//Note: the execution time is monitored by a base Fb timer. Therefore a timeout may occur. This behavior is configurable.
END_METHOD

METHOD PRIVATE FINAL M_FinishCommand
VAR 
	strLogMsg : STRING;	
END_VAR
IF localCmd.Control = cAbort AND bAbortionAllowed THEN		//Command was aborted by host
	localRes.Status := cFinAbrtd;

ELSIF localRes.Error = GVL.ERR_NO_ERROR THEN					//executed without error
	localRes.Status := cFinOk;
	
	//Log data
		M_Log(	LogLevel 	:= eLogLevel.TRACE, 
				strMethod 	:= 'M_FinishCommand',
				strLogMsg 	:= '|ADS - command finished successfully by SPS');	
ELSE
	localRes.Status := cFinErr;								//executed with error
	//Log data
		strLogMsg := CONCAT('|ADS - command finished faulty by SPS with ErrorId: ', WORD_TO_STRING(localRes.Error));
	
		M_Log(	LogLevel 	:= eLogLevel.TRACE, 
				strMethod 	:= 'M_FinishCommand',
				strLogMsg 	:= strLogMsg);				
END_IF

bCmdEnabledByIntern := TRUE;
eState := eCmdProcessing._RECEIVING;
END_METHOD

METHOD PROTECTED FINAL M_Log
VAR_INPUT
	strMethod 	: STRING(40);
	strLogMsg 	: STRING;
	LogLevel 	: eLogLevel;
END_VAR
VAR
	strCaller : STRING := 'FB_wCMD_Handler_Base.';
END_VAR
IF NOT GVL_AdsInterface.bLoggingOnOff_IncomingAds THEN 
	RETURN;
END_IF

strCaller := CONCAT(strInstanceName, '.');
strCaller := CONCAT(strCaller, strMethod);

//If Logging.prg is not available in project or to deactivate logging completely, just comment the following line out!
	Logging.Debug(strCaller, strLogMsg);
END_METHOD

METHOD PRIVATE FINAL M_ReceiveCommand
IF localCmd.Control = cRcv THEN
		
	//Delete result structure variable
		MEMSET(destaddr := ADR(localRes), fillbyte:=0, n:= SIZEOF(localRes));
		localres.ErrorComp 	:= wCompId;
		localres.Error 		:= GVL.ERR_NO_ERROR;
	
	//Set result struct to state RECEIVED even if there could be errors
		localRes.Status := cRcvd;
	
	//Check if command is currently blocked
	IF bCmdEnabledByExtern AND bCmdEnabledByIntern THEN
		bCmdEnabledByIntern := FALSE;
		
	ELSIF NOT bCmdEnabledByIntern THEN		
		localRes.Error := GVL_AdsInterface_ERROR_IDS.ERR_ITF_COMMAND_CAN_NOT_BE_ENABLED_THUS_INTERNALLY_DISABLED + GVL_AdsInterface.wErrorIdOffset_IncomingAds;
		
	ELSIF NOT bCmdEnabledByExtern THEN
		localRes.Error := GVL_AdsInterface_ERROR_IDS.ERR_ITF_COMMAND_CAN_NOT_BE_ENABLED_THUS_EXTERNALLY_DISABLED + GVL_AdsInterface.wErrorIdOffset_IncomingAds;
		
	ELSE
		localRes.Error := GVL_AdsInterface_ERROR_IDS.ERR_ITF_INCOMING_COMMAND_IS_BLOCKED + GVL_AdsInterface.wErrorIdOffset_IncomingAds;
		
	END_IF
	
	//Check incomming command parameter for correctness
		IF localCmd.Version 	<> wVersion 			THEN localRes.Error := GVL_AdsInterface_ERROR_IDS.ERR_ITF_INCOMING_COMMAND_HAS_WRONG_VERSION + GVL_AdsInterface.wErrorIdOffset_IncomingAds; 			END_IF;
		IF iParTyp 	<> PAR_TYPE_REGARDLESS THEN 
			IF localCmd.ParaCount 	<> iParCount 	THEN localRes.Error := GVL_AdsInterface_ERROR_IDS.ERR_ITF_INCOMING_COMMAND_HAS_WRONG_PARAMETER_COUNT + GVL_AdsInterface.wErrorIdOffset_IncomingAds; 	END_IF;
			IF localCmd.ParaTyp	 	<> iParTyp 		THEN localRes.Error := GVL_AdsInterface_ERROR_IDS.ERR_ITF_INCOMING_COMMAND_HAS_WRONG_PARAMETER_TYP + GVL_AdsInterface.wErrorIdOffset_IncomingAds; 	END_IF;				
		END_IF
END_IF
END_METHOD

PROPERTY PUBLIC final P_EnabledInternally : bool
GET
P_EnabledInternally := bCmdEnabledByIntern;
END_GET
END_PROPERTY

END_FUNCTION_BLOCK

// AdsInterface/FB_SendAdsDocCmd_Base
//Author: 				Walther Ronny
//Version:				1.0
//Last change:			14.04.16
//See Release notes at the bottom
//{attribute 'hide_all_locals'}
{attribute 'reflection'}
FUNCTION_BLOCK PUBLIC FB_SendAdsDocCmd_Base				//Base Fb for handling of ADS communication of type TwRes and TwCmd
VAR_OUTPUT
	bDone,
	bError : BOOL;
	ErrorMsg : sErrorMsg;
    {attribute 'instance-path'}
    {attribute 'no_init'}
    sPath  : STRING;
END_VAR 
VAR_INPUT		
	Instanz: BYTE; 										//Instanz counter 
	pCmd : POINTER TO TxCmdRes;							//Pointer to incomming command structure from host
	pRes : POINTER TO TxCmdRes;							//Pointer to outgoing result structure from SPS
END_VAR
VAR
	wCompId : WORD;		//Component ID
//Command configuration which has to be set by instantiated Fb - 	MUST !
	wVersion : 				WORD := 0;	//Expected version of incomming command
	iParTyp1: 				BYTE := 0;	//Expected parameter type of incomming command, PAR_TYPE_REGARDLESS will switch test off
	iParCount1 : 			BYTE := 0;	//Expected parameter count of incomming command
	iParTyp2 : 				BYTE := 0;	//Expected parameter type of incomming command, PAR_TYPE_REGARDLESS will switch test off
	iParCount2 : 			BYTE := 0;	//Expected parameter count of incomming command
	
//Command configuration which can be set by instantiated Fb - 	OPTIONALLY !
	tExecutionTimeout : 	TIME := ADS_EXECUTION_TIMEOUT; 	//Timeout while Execution running. T#0s equals off
	
	bStartSendingData : BOOL := FALSE;	//flag to indicate that data can be sent				

//This variable can be used to hold the state of the derived M_ExecuteCommand() 
	iHelpState : UINT := 0;	//optional help variable to create a statemachine inside derive M_ExecuteCommand()
	
//Local Command and result structure objects - Will be read and written by base Fb and derived "M_ExecuteCommand()" method
	localRes: TdocRes;
	localCmd: TdocCmd;	
	
//Internal variables of base Fb - DO NOT CHANGE!	
	bCmdEnabledByExtern,								//Command is enabled/disabled  externally (by MainFSM)
	bCmdEnabledByIntern : 	BOOL:= TRUE;				//Command is enabled/disabled  internally during execution
		
	eState: eSendCmdProcessing := eSendCmdProcessing._IDLE;	//Current internal state of the base Fb		
	TimerExecutionTimeout : ton;						// Timer for Execution timeout
END_VAR
VAR CONSTANT
	//Command parameter types
	PAR_TYPE_REGARDLESS :		BYTE := 0;			//if this type is set, the parameter type will be not checked
	PAR_TYPE_ANSICHAR : 		BYTE := 16#41;
	PAR_TYPE_SHORTINT : 		BYTE := 16#53;
	PAR_TYPE_WIDECHAR : 		BYTE := 16#43;
	PAR_TYPE_SMALLINT : 		BYTE := 16#4D;
	PAR_TYPE_LONGINT : 			BYTE := 16#49;
	PAR_TYPE_LONGWORD : 		BYTE := 16#4C;
	PAR_TYPE_WORD : 			BYTE := 16#57;		//Standard parameter type
	PAR_TYPE_BIT : 				BYTE := 16#58;
	
	ADS_EXECUTION_TIMEOUT :		TIME := T#10S;		//Timeout while derived Execution method is executed. T#0S equals OFF

		// command
	cAbort:						WORD := 0;			// command abort				
	cRcv:						WORD := 1;			// command receive				
	cExec:						WORD := 2;			// command start				
	// result
	cIdle: 						WORD := 0;      	// not  defined					
	cRcvd:						WORD := 1;      	// command received 			
	cActive:					WORD := 2;			// command active started 		
	cFinOk:						WORD := 4;			// command finished ok			
	cFinAbrtd:					WORD := 5;			// command aborted				
	cFinErr:					WORD := 6;			// command finished error		
END_VAR

(*
Release notes:
1.0 	Walther Ronny, 14.04.16
		- Initial version
*)

ErrorMsg.sFunctionName := 'FB_SendAdsDocCmd_Base';

	wCompId := GVL_AdsInterface.wCompId_OutgoingAds;
	
//Create local copy of actual result struct
	localRes := pRes^.docRes;

CASE eState OF
	
	eSendCmdProcessing._IDLE :
	
			//reset flags
				bError 	:= FALSE;
				bDone	:= FALSE;
				
			//reset timeout timer
				TimerExecutionTimeout.IN := FALSE;
				
			//Check for start sending flag	
				IF bStartSendingData THEN
					bStartSendingData := FALSE;
					
					//disable cmd
						bCmdEnabledByIntern := FALSE;
						
					//Set receive parameter
						localCmd.Control := cRcv;
						
					//Set local data to outgoing command struct					
						pCmd^.docCmd := localCmd;
					
					eState := eSendCmdProcessing._SENDING;
					Logging.Trace('FB_SendAdsDocCmd_Base','State change: IDLE - SENDING');
				END_IF
				
	eSendCmdProcessing._SENDING :
	
			IF localRes.Status = cRcvd THEN
				
				//Start command
					pCmd^.docCmd.Control := cExec;
					
				eState := eSendCmdProcessing._STARTING;
				Logging.Trace('FB_SendAdsDocCmd_Base','State change: SENDING - STARTING');
			END_IF
			
	eSendCmdProcessing._STARTING :
					
			//start timeout timer
				TimerExecutionTimeout(IN := TRUE, PT := tExecutionTimeout);
				
			//Wait for result state	to change
				IF localRes.Status <> cRcvd THEN				
					eState := eSendCmdProcessing._EXECUTING;
					Logging.Trace('FB_SendAdsDocCmd_Base','State change: STARTING - EXECUTING');
				END_IF
			
	eSendCmdProcessing._EXECUTING :
	
			IF localRes.Status = cFinOk THEN
				eState := eSendCmdProcessing._DONE;
				Logging.Trace('FB_SendAdsDocCmd_Base','State change: EXECUTING - DONE (cFinOK)');
			ELSIF localRes.Status = cFinAbrtd THEN
				bError 				:= TRUE;
				ErrorMsg.wComponent := wCompId;
				ErrorMsg.wErrorNo 	:= GVL_AdsInterface_ERROR_IDS.ERR_ITF_COMMAND_WAS_ABORTED_BY_HOST_DURING_EXECUTION + GVL_AdsInterface.wErrorIdOffset_OutgoingAds;
				
				eState := eSendCmdProcessing._DONE;
				Logging.Trace('FB_SendAdsDocCmd_Base','State change: EXECUTING - DONE (cFinAbrtd)');
			ELSIF localRes.Status = cFinErr THEN
				bError 				:= TRUE;
				ErrorMsg.wComponent := wCompId;
				ErrorMsg.wErrorNo 	:= localRes.Error + GVL_AdsInterface.wErrorIdOffset_OutgoingAds;
				
				eState := eSendCmdProcessing._DONE;
				Logging.Trace('FB_SendAdsDocCmd_Base','State change: EXECUTING - DONE (cFinErr)');
			ELSIF TimerExecutionTimeout.Q AND tExecutionTimeout <> T#0S THEN
				bError 				:= TRUE;
				ErrorMsg.wComponent := wCompId;
				ErrorMsg.wErrorNo 	:= GVL_AdsInterface_ERROR_IDS.ERR_ITF_COMMAND_EXECUTION_TIMEOUT + GVL_AdsInterface.wErrorIdOffset_OutgoingAds;
					
				eState := eSendCmdProcessing._DONE; 
				Logging.Trace('FB_SendAdsDocCmd_Base','State change: EXECUTING - DONE (timeout)');		
			END_IF
			
	eSendCmdProcessing._DONE : 
	
			//reset timeout timer
				TimerExecutionTimeout.IN := FALSE;
				
			bCmdEnabledByIntern := TRUE;
			
			bDone:= TRUE;
			
			//Check for start sending flag	
				IF bStartSendingData THEN
					eState := eSendCmdProcessing._IDLE;
					
				END_IF

END_CASE

TimerExecutionTimeout();

METHOD PUBLIC M_EnableCmd
VAR_INPUT
	bEnable : BOOL := FALSE; //TRUE = Command is enabled, FALSE = Command i disabled
END_VAR
bCmdEnabledByExtern := bEnable;
END_METHOD

METHOD PUBLIC M_SendCmd				//Sending an ADS command
VAR_INPUT
	docCmdData 		: TdocCmd; 		//command structure to be sent
END_VAR
VAR_OUTPUT
	bMethodError 	: BOOL;			//indicates an error
	MethodErrorMsg 	: sErrorMsg;	//describes an error
END_VAR
//Check command state
	IF eState = eSendCmdProcessing._IDLE OR eState = eSendCmdProcessing._DONE THEN
	
	//Reset fb output state
		bDone := FALSE;
		bError := FALSE;
		ErrorMsg.wComponent := wCompId;
		ErrorMsg.wErrorNo 	:= GVL.ERR_NO_ERROR;
		
		M_SetLocalData(pDocCmd := ADR(docCmdData), bError => bMethodError, ErrorMsg => MethodErrorMsg);
		
		IF NOT bMethodError THEN
			//start sending data
				bStartSendingData := TRUE;
				
		END_IF
		
	ELSE //e.g. still activ...
		bMethodError := TRUE;
		MethodErrorMsg.wComponent := wCompId;
		MethodErrorMsg.wErrorNo	:= GVL_AdsInterface_ERROR_IDS.ERR_ITF_WRONG_FB_STATE_TO_SEND_COMMAND + GVL_AdsInterface.wErrorIdOffset_OutgoingAds;
		
	END_IF
END_METHOD

METHOD PRIVATE M_SetLocalData
VAR_INPUT
	pDocCmd : pointer to TdocCmd;
END_VAR
VAR_OUTPUT
	bError : 	BOOL;
	ErrorMsg : 	sErrorMsg;
END_VAR
	//Delete result structure variable
		MEMSET(destaddr := ADR(localRes), fillbyte:=0, n:= SIZEOF(localRes));
	
	//Check if command is currently blocked
	IF bCmdEnabledByExtern AND bCmdEnabledByIntern THEN
		ErrorMsg.wErrorNo := GVL.ERR_NO_ERROR;
		bCmdEnabledByIntern := FALSE;
		
	ELSIF NOT bCmdEnabledByIntern THEN		
		ErrorMsg.wErrorNo := GVL_AdsInterface_ERROR_IDS.ERR_ITF_COMMAND_CAN_NOT_BE_ENABLED_THUS_INTERNALLY_DISABLED + GVL_AdsInterface.wErrorIdOffset_OutgoingAds;
		
	ELSIF NOT bCmdEnabledByExtern THEN
		ErrorMsg.wErrorNo := GVL_AdsInterface_ERROR_IDS.ERR_ITF_COMMAND_CAN_NOT_BE_ENABLED_THUS_EXTERNALLY_DISABLED + GVL_AdsInterface.wErrorIdOffset_OutgoingAds;
		
	ELSE
		ErrorMsg.wErrorNo := GVL_AdsInterface_ERROR_IDS.ERR_ITF_INCOMING_COMMAND_IS_BLOCKED + GVL_AdsInterface.wErrorIdOffset_OutgoingAds;
		
	END_IF
	
	//Check incomming command parameter for correctness
		IF pDocCmd^.Version 	<> wVersion 			THEN ErrorMsg.wErrorNo := GVL_AdsInterface_ERROR_IDS.ERR_ITF_INCOMING_COMMAND_HAS_WRONG_VERSION + GVL_AdsInterface.wErrorIdOffset_OutgoingAds; 		END_IF;
			
		IF iParTyp1 	<> PAR_TYPE_REGARDLESS 	THEN 
			IF pDocCmd^.ParaCount1 	<> iParCount1 	THEN ErrorMsg.wErrorNo := GVL_AdsInterface_ERROR_IDS.ERR_ITF_INCOMING_COMMAND_HAS_WRONG_PARAMETER_COUNT + GVL_AdsInterface.wErrorIdOffset_OutgoingAds; 	END_IF;
			IF pDocCmd^.ParaTyp1	<> iParTyp1		THEN ErrorMsg.wErrorNo := GVL_AdsInterface_ERROR_IDS.ERR_ITF_INCOMING_COMMAND_HAS_WRONG_PARAMETER_TYP + GVL_AdsInterface.wErrorIdOffset_OutgoingAds; 	END_IF;	
		END_IF;	
		
		IF iParTyp2 	<> PAR_TYPE_REGARDLESS THEN
			IF pDocCmd^.ParaCount2 	<> iParCount2 	THEN ErrorMsg.wErrorNo := GVL_AdsInterface_ERROR_IDS.ERR_ITF_INCOMING_COMMAND_HAS_WRONG_PARAMETER_COUNT + GVL_AdsInterface.wErrorIdOffset_OutgoingAds; 	END_IF;			
			IF pDocCmd^.ParaTyp2	<> iParTyp2		THEN ErrorMsg.wErrorNo := GVL_AdsInterface_ERROR_IDS.ERR_ITF_INCOMING_COMMAND_HAS_WRONG_PARAMETER_TYP + GVL_AdsInterface.wErrorIdOffset_OutgoingAds; 	END_IF;	
		END_IF
	ErrorMsg.wComponent := wCompId;
	
	IF ErrorMsg.wErrorNo <> GVL.ERR_NO_ERROR THEN
		bError:= TRUE;
	ELSE
		localCmd := pDocCmd^;	

	END_IF
END_METHOD

PROPERTY PUBLIC P_CommandState : eSendCmdProcessing
GET
P_CommandState := eState;
END_GET
END_PROPERTY

PROPERTY PUBLIC P_EnabledInternally : bool
GET
P_EnabledInternally := bCmdEnabledByIntern;
END_GET
END_PROPERTY

END_FUNCTION_BLOCK

// AdsInterface/FB_wCMD_docCMD_Handler_Base2
//Author: 				Walther Ronny
//Version:				1.6
//Last change:			16.10.2018
//See Release notes at the bottom
//{attribute 'hide_all_locals'}
{attribute 'reflection'}
FUNCTION_BLOCK PUBLIC FB_wCMD_docCMD_Handler_Base2				//Base Fb for handling of ADS communication of type TwRes and TwCmd
VAR_OUTPUT
    {attribute 'instance-path'}
    {attribute 'no_init'}
    sPath  		: STRING; 	//Instance path
	pLogCmdRes 	: POINTER TO ARRAY [0.. LOG_CMDRES_MAX] OF TxCmdRes2Double := ADR(arrLogCmdRes);
	pLogCmdResIndex: POINTER TO UINT := ADR(nLogIndexCmdRes);
END_VAR 
VAR_INPUT		
	Instanz: BYTE; 										//Instanz counter 
	pCmd : POINTER TO TxCmdRes2;						//Pointer to incomming command structure from host
	pRes : POINTER TO TxCmdRes2;						//Pointer to outgoing result structure from SPS
END_VAR
VAR		
	wCompId : WORD;		//Component ID
//Command configuration which has to be set by instantiated Fb - 	MUST !
	wVersion : 				WORD := 0;	//Expected version of incomming command
	iParTyp1 : 				BYTE := 0;	//Expected parameter type of incomming command, PAR_TYPE_REGARDLESS will switch test off
	iParCount1 : 			BYTE := 0;	//Expected parameter count of incomming command
	iParTyp2 : 				BYTE := 0;	//Expected parameter type of incomming command, PAR_TYPE_REGARDLESS will switch test off
	iParCount2 : 			BYTE := 0;	//Expected parameter count of incomming command
		
//Command configuration which can be set by instantiated Fb - 	OPTIONALLY !
	bAbortionAllowed : 		BOOL 		:= TRUE;					//if yes, abortion from host is allowed all the time
	tExecutionTimeout : 	TIME 		:= ADS_EXECUTION_TIMEOUT; 	//Timeout while Execution running. T#0s equals off
	strInstanceName :		STRING(40);								//Name of instance of that base class (used only for logging purposes)
//Flag to indicate that the derived method "M_ExecuteCommand()" finished	
	bExecutionDone : BOOL := FALSE;	//flag to indicate that derived Execution is done				

//This variable can be used to hold the state of the derived M_ExecuteCommand() 
	iHelpState : UINT := 0;	//optional help variable to create a statemachine inside derive M_ExecuteCommand()
	
//Local Command and result structure objects - Will be read and written by base Fb and derived "M_ExecuteCommand()" method
	localRes: TxCmdRes2;//TwRes2;
	localCmd: TxCmdRes2;//TwCmd2;	
	
//Internal variables of base Fb - DO NOT CHANGE!	
	bCmdEnabledByExtern,								//Command is enabled/disabled  externally (by MainFSM)
	bCmdEnabledByIntern : 	BOOL:= TRUE;				//Command is enabled/disabled  internally during execution
		
	eState: eCmdProcessing := eCmdProcessing._RECEIVING;	//Current internal state of the base Fb		
	TimerExecutionTimeout : ton;							// Timer for Execution timeout
	
// log ads communication for debugging	
	nCmpResult, nCmpCommand: DINT;
	nLogIndexCmdRes: UINT;
	arrLogCmdRes: ARRAY [0.. LOG_CMDRES_MAX] OF TxCmdRes2Double;
	
	
END_VAR
VAR CONSTANT
	LOG_CMDRES_MAX:				UINT := 10;
	DATA_LENGT_IN_8byte:		UINT := 7;	

	//Command parameter types
	PAR_TYPE_REGARDLESS :		BYTE := 0;		//if this type is set, the parameter type will be not checked
	PAR_TYPE_ANSICHAR : 		BYTE := 16#41; //8bit
	PAR_TYPE_BYTE : 			BYTE := 16#42; //8bit
	PAR_TYPE_WIDECHAR : 		BYTE := 16#43; //16bit
	PAR_TYPE_FLOAT : 			BYTE := 16#44; //64bit	
	PAR_TYPE_SHORTINT : 		BYTE := 16#53; //8bit	
	PAR_TYPE_SMALLINT : 		BYTE := 16#4D; //16bit
	PAR_TYPE_LONGINT : 			BYTE := 16#49; //32bit
	PAR_TYPE_LONGWORD : 		BYTE := 16#4C; //32bit
	PAR_TYPE_WORD : 			BYTE := 16#57; //16bit
	PAR_TYPE_BIT : 				BYTE := 16#58;
	
	ADS_EXECUTION_TIMEOUT :		TIME := T#30S;		//Timeout while derived Execution method is executed. T#0S equals OFF

		// command
	cAbort:						WORD := 0;			// command abort				
	cRcv:						WORD := 1;			// command receive				
	cExec:						WORD := 2;			// command start				
	// result
	cIdle: 						WORD := 0;      	// not  defined					
	cRcvd:						WORD := 1;      	// command received 			
	cActive:					WORD := 2;			// command active started 		
	cFinOk:						WORD := 4;			// command finished ok			
	cFinAbrtd:					WORD := 5;			// command aborted				
	cFinErr:					WORD := 6;			// command finished error		
END_VAR

(*
Release notes:
1.0 First release. Tested on Holo machine in Munich. 25.01.16
1.1 Aborting modified and tested. Constants included in FB. 26.01.16
1.2 Bug M_ReceiveCommand PARTYP_REGARDLESS fixed
1.3 Walther Ronny, 25.05.16
	- Variable strInstanceName added
	- Method M_Log() added
	- Logging added
1.4 Werner Richter, 19.09.2018
	- FB_wCMD_Handler_Base modifyed to FB_wCMD_Handler_Base2 because communication to host has modified to check data length before sending,
	  use modified data structure TxCmdRes2, check header in state _RECEIVING, modify M_ReceiveCommand, 
      check type in _WAITING_FOR_START, set received flag only if no error
1.5 Werner Richter, 21.09.2018
	- combined FB_wCMD_Handler_Base2 + FB_docCMD_Handler_Base, bAbortionAllowed := TRUE
1.6 Werner Richter, 16.10.2018
	- log ads communication for debugging
*)

//Create local copy of received command struct
	localCmd:=pCmd^;//.wCmd; 

CASE eState OF
	
	eCmdProcessing._RECEIVING: 	//Receiving command
	
				//Check id, thus it might have been changed
					wCompId := GVL_AdsInterface.wCompId_IncomingAds;
				
				IF M_ReceiveCommand() THEN
								
					//Log data
					M_Log(	LogLevel 	:= eLogLevel.TRACE, 
							strMethod 	:= 'FB_wCMD_Handler_Base',
							strLogMsg 	:= '|ADS - command received from host');	
								
					IF localres.wRes.Error = GVL.ERR_NO_ERROR THEN	// check wrong header
								
						localRes.wRes.Status := cRcvd;
						eState := eCmdProcessing._WAITING_FOR_START;					
					ELSE
						
						localRes.wRes.Status := cFinErr;
						
						pCmd^.wCmd.Control := cAbort;			// needed if error in receiving state occured to reset command handshaking
	
						//Log data					
						M_Log(	LogLevel 	:= eLogLevel.TRACE, 
								strMethod 	:= 'M_FinishCommand',
								strLogMsg 	:= CONCAT('|ADS - command finished faulty by SPS with ErrorId: ', WORD_TO_STRING(localRes.wRes.Error)));				
										
						bCmdEnabledByIntern := TRUE;
						eState := eCmdProcessing._RECEIVING;
						
						//reset timer
						TimerExecutionTimeout.IN := FALSE;						
						
					END_IF
					
				END_IF
								
							
				
	eCmdProcessing._WAITING_FOR_START:	//Waiting for Start from Host
					
				IF localCmd.wCmd.Control = cExec THEN //check if the command was started by the host
					//Log data
						M_Log(	LogLevel 	:= eLogLevel.TRACE, 
								strMethod 	:= 'FB_wCMD_Handler_Base',
								strLogMsg 	:= '|ADS - command started by host');	
						
								
					IF localRes.wRes.Error <> GVL.ERR_NO_ERROR THEN //Check if an error during receiving ocurred		
	
						eState := eCmdProcessing._FINISHING;

					ELSIF 	((iParTyp1 <> PAR_TYPE_REGARDLESS) AND ((localCmd.wCmd.ParaCount1 <> iParCount1) OR (localCmd.wCmd.ParaTyp1 <> iParTyp1))) OR
							((iParTyp2 <> PAR_TYPE_REGARDLESS) AND ((localCmd.docCmd.ParaCount2 <> iParCount2) OR (localCmd.docCmd.ParaTyp2 <> iParTyp2))) THEN
					
						// wCmd	+ docCmd	
						IF (iParTyp1 <> PAR_TYPE_REGARDLESS) AND ((localCmd.wCmd.ParaCount1 <> iParCount1) OR (localCmd.wCmd.ParaTyp1 <> iParTyp1)) THEN										
							IF localCmd.wCmd.ParaCount1 <> iParCount1 THEN localRes.wRes.Error := GVL_AdsInterface_ERROR_IDS.ERR_ITF_INCOMING_COMMAND_HAS_WRONG_PARAMETER_COUNT + GVL_AdsInterface.wErrorIdOffset_IncomingAds; 	END_IF;
							IF localCmd.wCmd.ParaTyp1   <> iParTyp1   THEN localRes.wRes.Error := GVL_AdsInterface_ERROR_IDS.ERR_ITF_INCOMING_COMMAND_HAS_WRONG_PARAMETER_TYP + GVL_AdsInterface.wErrorIdOffset_IncomingAds; 	END_IF;										
						END_IF
						
						//docCmd
						IF (iParTyp2 <> PAR_TYPE_REGARDLESS) AND ((localCmd.docCmd.ParaCount2 <> iParCount2) OR (localCmd.docCmd.ParaTyp2 <> iParTyp2)) THEN							
							IF localCmd.docCmd.ParaCount2 <> iParCount2 THEN localRes.wRes.Error := GVL_AdsInterface_ERROR_IDS.ERR_ITF_INCOMING_COMMAND_HAS_WRONG_PARAMETER_COUNT + GVL_AdsInterface.wErrorIdOffset_IncomingAds; 	END_IF;
							IF localCmd.docCmd.ParaTyp2	  <> iParTyp2   THEN localRes.wRes.Error := GVL_AdsInterface_ERROR_IDS.ERR_ITF_INCOMING_COMMAND_HAS_WRONG_PARAMETER_TYP + GVL_AdsInterface.wErrorIdOffset_IncomingAds; 	END_IF;										
						END_IF
						
						eState := eCmdProcessing._FINISHING;

					ELSE
																									
						//Reset variables for derived "M_ExecuteCommand()" method	
							bExecutionDone := FALSE;
							iHelpState := 0;	
						
						localRes.wRes.Status := cActive;					
						eState := eCmdProcessing._EXECUTING;
						
						//start timeout timer
							TimerExecutionTimeout(IN := TRUE, PT := tExecutionTimeout);
					END_IF					
								
					
				END_IF
					
					
	eCmdProcessing._EXECUTING:	//Executing command
			
				IF bExecutionDone THEN //flag will be set by derived method if execution done									
					eState := eCmdProcessing._FINISHING; 
					
				ELSIF TimerExecutionTimeout.Q AND tExecutionTimeout <> T#0S THEN
					localRes.wRes.ErrorComp := wCompId;	
					localRes.wRes.Error := GVL_AdsInterface_ERROR_IDS.ERR_ITF_COMMAND_EXECUTION_TIMEOUT + GVL_AdsInterface.wErrorIdOffset_IncomingAds;
					
					eState := eCmdProcessing._FINISHING; 			
					
				ELSE //derived method will be executed
					M_ExecuteCommand();
						
				END_IF
	
		
	eCmdProcessing._FINISHING: //Finishing Command
		
				M_FinishCommand();
				
				//reset timer
					TimerExecutionTimeout.IN := FALSE;
				
				
	eCmdProcessing._ABORTING: //Aborting Command
				
				eState := eCmdProcessing._FINISHING; 
				
END_CASE

//check if aborted by host and command configured "bAbortionAllowed
//Note: 	Thus abortion is possible all the time the execution could be interuppted at an unsafe state!
//			Preferable abortion should be allowed only for service commands which a triggered manually from an operator.
	IF localCmd.wCmd.Control = cAbort AND bAbortionAllowed 
		AND eState <> eCmdProcessing._ABORTING 		//Not allowed cause aborting already active
		AND eState <> eCmdProcessing._FINISHING 	//Not allowed cause command is finishing anyway
		AND eState <> eCmdProcessing._RECEIVING		//Not allowed cause command have not been started yet
		THEN 
			
			IF eState = eCmdProcessing._EXECUTING THEN  //cause eventually leaving unsafe state, throw error
				localRes.wRes.ErrorComp := wCompId;	
				localRes.wRes.Error := GVL_AdsInterface_ERROR_IDS.ERR_ITF_COMMAND_WAS_ABORTED_BY_HOST_DURING_EXECUTION + GVL_AdsInterface.wErrorIdOffset_IncomingAds;
				
			END_IF
			
			eState := eCmdProcessing._ABORTING;
			
	END_IF
	

TimerExecutionTimeout();

pRes^ := localRes;


A_LogResChanges();

ACTION A_LogResChanges:
// Author: 				Werner Richter
// Version:				1.00
// Last change:			16.10.2018
// See Release notes at the bottom

// log ads communication for debugging

	nCmpCommand := MEMCMP(ADR(arrLogCmdRes[nLogIndexCmdRes].Cmd), pCmd, SIZEOF(TxCmdRes2));
	nCmpResult := MEMCMP(ADR(arrLogCmdRes[nLogIndexCmdRes].Res), pRes, SIZEOF(TxCmdRes2));
	
	// check if Res struct was changing
	IF ((nCmpResult <> 0) OR (nCmpCommand <> 0)) THEN	
		
		IF nLogIndexCmdRes < LOG_CMDRES_MAX THEN
			nLogIndexCmdRes := nLogIndexCmdRes + 1;
		ELSE
			nLogIndexCmdRes := 0;
		END_IF
		
		arrLogCmdRes[nLogIndexCmdRes].Cmd := pCmd^;		
		arrLogCmdRes[nLogIndexCmdRes].Res := pRes^;	

	END_IF

(*
V1.00 Werner Richter, 16.10.2018
		- initial version 
*)
END_ACTION

METHOD PUBLIC FINAL M_EnableCmd
VAR_INPUT
	bEnable : BOOL := FALSE; //TRUE = Command is enabled, FALSE = Command i disabled
END_VAR
bCmdEnabledByExtern := bEnable;
END_METHOD

METHOD PUBLIC M_ExecuteCommand // to be derived and customized....
// to be derived and customized....



//To DO`s of the derived Method:
 
//1. Check Data for correctness
//2. set optional result data 
//3. iHelpState vaiable can be used
//4. if an Error occured localRes.Error and localRes.ErrorComp has to be set!
//5. at last the "bExecutionDone" flag has to be set. This will start the transition to the M_FinishCommand Method inside the base FB.

//Note: the execution time is monitored by a base Fb timer. Therefore a timeout may occur. This behavior is configurable.
END_METHOD

METHOD PRIVATE FINAL M_FinishCommand
VAR 
	strLogMsg : STRING;	
END_VAR
IF localCmd.wCmd.Control = cAbort AND bAbortionAllowed THEN		//Command was aborted by host
	localRes.wRes.Status := cFinAbrtd;

ELSIF localRes.wRes.Error = GVL.ERR_NO_ERROR THEN				//executed without error
	localRes.wRes.Status := cFinOk;
	
	//Log data
		M_Log(	LogLevel 	:= eLogLevel.TRACE, 
				strMethod 	:= 'M_FinishCommand',
				strLogMsg 	:= '|ADS - command finished successfully by SPS');	
ELSE
	
	//pCmd^.wCmd.Control := cAbort;							// needed if error in receiving state occured to reset command handshaking

	localRes.wRes.Status := cFinErr;								//executed with error
	//Log data
		strLogMsg := CONCAT('|ADS - command finished faulty by SPS with ErrorId: ', WORD_TO_STRING(localRes.wRes.Error));
	
		M_Log(	LogLevel 	:= eLogLevel.TRACE, 
				strMethod 	:= 'M_FinishCommand',
				strLogMsg 	:= strLogMsg);				
END_IF

bCmdEnabledByIntern := TRUE;
eState := eCmdProcessing._RECEIVING;
END_METHOD

METHOD PROTECTED FINAL M_Log
VAR_INPUT
	strMethod 	: STRING(40);
	strLogMsg 	: STRING;
	LogLevel 	: eLogLevel;
END_VAR
VAR
	strCaller : STRING := 'FB_wCMD_Handler_Base.';
END_VAR
IF NOT GVL_AdsInterface.bLoggingOnOff_IncomingAds THEN 
	RETURN;
END_IF

strCaller := CONCAT(strInstanceName, '.');
strCaller := CONCAT(strCaller, strMethod);

//If Logging.prg is not available in project or to deactivate logging completely, just comment the following line out!
	Logging.Debug(strCaller, strLogMsg);
END_METHOD

METHOD PRIVATE FINAL M_ReceiveCommand : BOOL;
IF localCmd.wCmd.Control = cRcv THEN
		
	//Delete result structure variable
		MEMSET(destaddr := ADR(localRes), fillbyte:=0, n:= SIZEOF(localRes));
		localres.wRes.ErrorComp 	:= wCompId;
		localres.wRes.Error 		:= GVL.ERR_NO_ERROR;
	
	//Set result struct to state RECEIVED even if there could be errors -> not with new structure!
	//	localRes.Status := cRcvd;
	
	//Check if command is currently blocked
	IF bCmdEnabledByExtern AND bCmdEnabledByIntern THEN
		bCmdEnabledByIntern := FALSE;
		
	ELSIF NOT bCmdEnabledByIntern THEN		
		localRes.wRes.Error := GVL_AdsInterface_ERROR_IDS.ERR_ITF_COMMAND_CAN_NOT_BE_ENABLED_THUS_INTERNALLY_DISABLED + GVL_AdsInterface.wErrorIdOffset_IncomingAds;
		
	ELSIF NOT bCmdEnabledByExtern THEN
		localRes.wRes.Error := GVL_AdsInterface_ERROR_IDS.ERR_ITF_COMMAND_CAN_NOT_BE_ENABLED_THUS_EXTERNALLY_DISABLED + GVL_AdsInterface.wErrorIdOffset_IncomingAds;
		
	ELSE
		localRes.wRes.Error := GVL_AdsInterface_ERROR_IDS.ERR_ITF_INCOMING_COMMAND_IS_BLOCKED + GVL_AdsInterface.wErrorIdOffset_IncomingAds;
		
	END_IF
	
	//Check incomming command parameter for correctness
	IF localCmd.wCmd.Version <> wVersion THEN 
		localRes.wRes.Error := GVL_AdsInterface_ERROR_IDS.ERR_ITF_INCOMING_COMMAND_HAS_WRONG_VERSION + GVL_AdsInterface.wErrorIdOffset_IncomingAds; 	
	
	ELSIF localCmd.wCmd.CmdDataLengthIn8Byte <> DATA_LENGT_IN_8byte THEN		
		localRes.wRes.Error := GVL_AdsInterface_ERROR_IDS.ERR_ITF_INCOMING_COMMAND_HAS_WRONG_COMMAND_DATA_SIZE + GVL_AdsInterface.wErrorIdOffset_IncomingAds; 
		
	ELSIF localCmd.wCmd.ResDataLengthIn8Byte <> DATA_LENGT_IN_8byte THEN
		
		localRes.wRes.Error := GVL_AdsInterface_ERROR_IDS.ERR_ITF_INCOMING_COMMAND_HAS_WRONG_RESULT_DATA_SIZE + GVL_AdsInterface.wErrorIdOffset_IncomingAds; 
	END_IF;

	M_ReceiveCommand := TRUE;
	

END_IF
END_METHOD

PROPERTY PUBLIC final P_EnabledInternally : bool
GET
P_EnabledInternally := bCmdEnabledByIntern;
END_GET
END_PROPERTY

END_FUNCTION_BLOCK

// AdsInterface/InitializeAds_Incoming
FUNCTION InitializeAds_Incoming : bool
VAR_INPUT
	wCompId 		: tErrorConstant;	//TRUE => Logging activated, FALSE => Logging deactivated
	wErrorIdOffset	: tErrorConstant;	//Offset to be added to all ErrorId´s	
	bLoggingOnOff 	: BOOL;				//TRUE => Logging activated, FALSE => Logging deactivated
END_VAR
VAR
END_VAR

GVL_AdsInterface.wCompId_IncomingAds 		:= wCompId;
GVL_AdsInterface.wErrorIdOffset_IncomingAds := wErrorIdOffset;
GVL_AdsInterface.bLoggingOnOff_IncomingAds	:= bLoggingOnOff;

InitializeAds_Incoming := TRUE;

END_FUNCTION

// AdsInterface/InitializeAds_Outgoing
FUNCTION InitializeAds_Outgoing : bool
VAR_INPUT
	wCompId 		: tErrorConstant;	//TRUE => Logging activated, FALSE => Logging deactivated
	wErrorIdOffset	: tErrorConstant;	//Offset to be added to all ErrorId´s	
	bLoggingOnOff 	: BOOL;				//TRUE => Logging activated, FALSE => Logging deactivated
END_VAR
VAR
END_VAR

GVL_AdsInterface.wCompId_OutgoingAds 			:= wCompId;
GVL_AdsInterface.wErrorIdOffset_OutgoingAds 	:= wErrorIdOffset;
GVL_AdsInterface.bLoggingOnOff_OutgoingAds		:= bLoggingOnOff;

InitializeAds_Outgoing := TRUE;

END_FUNCTION

// DocManagement/DocManagement
//Author: 				Koster Daniel, Walther Ronny
//Version:				1.4
//Last change:			14.04.16
//See Release notes at the bottom

PROGRAM DocManagement

VAR CONSTANT
	DOC_ARRAY_SIZE:			UINT:= 1000; //{warning 'RON - doc array temporarly huge!'}
	EMPTY_DOC : sDocument := (	Free 			:= TRUE, 		
								ID 				:= 0,
						 		Module 			:= 0,
								Location 		:= 0, 		
								Path 			:= 0, 
								PositionIndex	:= eDocPositionIndex.UNDEFINED,		
								Released 		:= TRUE,
								bReleaseHandshakeActive := TRUE,
								bLockedBySps 	:= FALSE,
								Moving 			:= FALSE,	
								Error 			:= FALSE);
END_VAR
VAR
	DocList:			ARRAY[0..(DOC_ARRAY_SIZE-1)] OF sDocument;
END_VAR
VAR_OUTPUT
	bDocsInBuffer: BOOL;
END_VAR

(*
V1.0 Koster Daniel
		- initial version
V1.1 Walther Ronny, 26.01.16 complete rework:
		- see release notes inside method deklaration
V1.2 Walther Ronny, 03.03.16 complete rework:
		- eDocPositionIndex hinzugefügt
V1.3 Walther Ronny, 14.03.16 complete rework:
		- bReleaseHandshakeActive implemented 
V1.4 Walther Ronny, 14.04.16 minor change:
		- EMPTY_DOC as constant instead var
*)

METHOD PUBLIC M_CheckDocsInPrevLocation
VAR_INPUT
	iCurLocation : UINT;
END_VAR
VAR_OUTPUT
	iDocsInPreviousLocation : UINT := 0;
	iSmallestID : UDINT;
END_VAR
VAR
	i:UINT;
END_VAR
(*
V1.0  Walther Ronny, 23.12.15
		- initial version
*)
iSmallestID := 16#FFFF;	
		
		//Count docs in previous location and find their smallest ID
		FOR i := 0 TO (DOC_ARRAY_SIZE - 1) DO
		
			IF NOT DocList[i].Free AND DocList[i].Location = iCurLocation-1 THEN
				
				iDocsInPreviousLocation := iDocsInPreviousLocation + 1;
				
				IF iSmallestID > DocList[i].ID THEN
					iSmallestID := DocList[i].ID;
				END_IF
			END_IF
	
		END_FOR
END_METHOD

METHOD public M_FindDoc
VAR_INPUT
	iDocID : UDINT;
END_VAR
VAR_OUTPUT
	bDocFound : 		BOOL := FALSE;
	pDoc : 				POINTER TO sDocument; //pointer to found document
	bMethodError : 		BOOL := FALSE;
	MethodErrorMsg : 	sErrorMsg;
END_VAR
VAR
	i : UINT;
END_VAR
(*
V1.0  Walther Ronny, 23.12.15
		- initial version, check if free
*)
MethodErrorMsg.wComponent 		:= GVL_DocManagement.wCompId;
MethodErrorMsg.sFunctionName 	:= 'M_GetDocInfoById';
MethodErrorMsg.wErrorNo 		:= GVL.ERR_NO_ERROR;

IF iDocID = 0 THEN
	bMethodError 				:= TRUE;			
	MethodErrorMsg.wErrorNo 	:= GVL_DocManagement_ERROR_IDS.ERR_DOC_ID_ZERO_INVALID + GVL_DocManagement.wErrorIdOffset;
	
ELSE
	//Find doc
	 FOR i := 0 TO (DOC_ARRAY_SIZE - 1) DO
					
		IF DocList[i].ID = iDocID AND NOT bDocFound AND NOT DocList[i].Free THEN
			pDoc := ADR(DocList[i]);
			bDocFound := TRUE;
			
		END_IF
					
	END_FOR
END_IF
END_METHOD

METHOD PUBLIC M_GetDocArrayInformation
VAR_OUTPUT
	iDocCount,
	iNumOfLockedDocs,
	iNumOfUnReleasedDocs,
	iNumOfDocsInLocationZero,
	iFreeSpaceCount :		UINT := 0;
		
	iSmallestDocId,
	iHighestDocId :			UDINT := 0;
	
	iLastFreeArrayIndex	 :	UINT := 0;
	
	bMethodError : 			BOOL := FALSE;
	MethodErrorMsg : 		sErrorMsg;
END_VAR
VAR
	i : UINT;
END_VAR
(*
V1.0  Walther Ronny, 27.12.15
		- initial version
*)
MethodErrorMsg.wComponent 		:= GVL_DocManagement.wCompId;
MethodErrorMsg.sFunctionName 	:= 'M_GetDocArrayInformation';
MethodErrorMsg.wErrorNo 		:= GVL.ERR_NO_ERROR;

	//Find doc
	 FOR i := 0 TO (DOC_ARRAY_SIZE - 1) DO
		
		IF DocList[i].Free THEN
			//Determine free spaces
		 		iFreeSpaceCount := iFreeSpaceCount +1;
				
			//Determine last free array index
				iLastFreeArrayIndex := i;
		ELSE
			//Count docs
				iDocCount := iDocCount + 1;
				
			//Determine highest ID
				IF DocList[i].ID >	iHighestDocId THEN
					iHighestDocId := DocList[i].ID;
				END_IF
			
			//Determine smallest ID	
				IF DocList[i].ID < iSmallestDocId OR iSmallestDocId = 0 THEN
					iSmallestDocId := DocList[i].ID;
				END_IF
				
			//Determine Num of locked docs
				IF DocList[i].bLockedBySps THEN
					iNumOfLockedDocs := iNumOfLockedDocs + 1;
				END_IF
				
			//Determine Num of unreleased docs
				IF NOT DocList[i].Released THEN
					iNumOfUnReleasedDocs := iNumOfUnReleasedDocs + 1;
				END_IF
				
			//Determine Num of docs in location 0 (=buffer and ready to be processed)
				IF DocList[i].Location = 0 THEN
					iNumOfDocsInLocationZero := iNumOfDocsInLocationZero + 1;
				END_IF
				
				
		END_IF
			

					
	END_FOR
END_METHOD

METHOD M_GetDocInfoById : sDocument
VAR_INPUT
	ID:			UDINT;
END_VAR
VAR_OUTPUT
	bDocFound : 		BOOL := FALSE;
	bMethodError : 		BOOL := FALSE;
	MethodErrorMsg : 	sErrorMsg;
END_VAR
VAR
	i : 				UINT;
	pDoc : 				POINTER TO sDocument;
	FoundDoc : 			sDocument;
	bDocIdFound : 		BOOL := FALSE;
END_VAR
(*
V1.0 Koster Daniel
		- initial version
V1.1 Walther Ronny, 26.01.16 major rework:
		- sErrorMsg integrated
		- unique Error IDs added
		- setting Done, Error flag in mother FB removed
		- no error, if not found but result flag
*)
MethodErrorMsg.wComponent 		:= GVL_DocManagement.wCompId;
MethodErrorMsg.sFunctionName 	:= 'M_GetDocInfoById';
MethodErrorMsg.wErrorNo 		:= GVL.ERR_NO_ERROR;

//just check if doc id exists
	M_FindDoc(iDocId := ID, bDocFound => bDocFound, pDoc => pDoc, bMethodError => bMethodError, MethodErrorMsg => MethodErrorMsg);
	
IF NOT bMethodError THEN
	IF bDocFound THEN
		FoundDoc := pDoc^;	//Document found 	
	
	ELSE
		bMethodError := TRUE;		
		MethodErrorMsg.wErrorNo := GVL_DocManagement_ERROR_IDS.ERR_DOC_ID_DOES_NOT_EXIST + GVL_DocManagement.wErrorIdOffset;
	
	END_IF
END_IF
M_GetDocInfoById := FoundDoc;
END_METHOD

METHOD PUBLIC M_Initialize
VAR_INPUT
	wCompId 			: tErrorConstant;		//TRUE => Logging activated, FALSE => Logging deactivated
	wErrorIdOffset		: tErrorConstant;		//Offset to be added to all ErrorId´s

END_VAR
GVL_DocManagement.wCompId 			:= wCompId;
GVL_DocManagement.wErrorIdOffset 	:= wErrorIdOffset;
END_METHOD

METHOD M_InsertNewDoc
VAR_INPUT
	ID:				UDINT;
	Module:			UINT;
	Location:		UINT; 
	Path:			UINT;
	RedAtLocation:	UINT;
	RedToLocation:	UINT;
	bReleaseHandshakeActive: BOOL; 
END_VAR
VAR_OUTPUT
	iDocIdSet : UDINT := 0;
	bMethodError : BOOL := FALSE;
	MethodErrorMsg : sErrorMsg;
END_VAR
VAR
	i : UINT;
	bDocIdExisting : BOOL := FALSE;
	
	iDocCount,
	iFreeSpaceCount :	UINT := 0;

	iLastFreeArrayIndex :	UINT := 0;	
	iSmallestDocId,
	iHighestDocId :		UDINT := 0;
END_VAR
(*
V1.0 Koster Daniel
		- initial version
V1.1 Walther Ronny, 26.01.16 complete rework:
		- sErrorMsg integrated
		- unique Error IDs added
		- setting Done, Error flag in mother FB removed
		- error checks modified, added
		- ID = 0 forces SPS to define a DocID
V1.2	Walther Ronny, 29.01.16
		-standard released value changed to TRUE
*)
MethodErrorMsg.wComponent 		:= GVL_DocManagement.wCompId;
MethodErrorMsg.sFunctionName 	:= 'M_InsertNewDoc';
MethodErrorMsg.wErrorNo 		:= GVL.ERR_NO_ERROR;

//Gather actual information
	M_GetDocArrayInformation(	iDocCount 			=> iDocCount,
								iFreeSpaceCount 	=> iFreeSpaceCount,
								iSmallestDocId 		=> iSmallestDocId,
								iHighestDocId 		=> iHighestDocId,
								iLastFreeArrayIndex => iLastFreeArrayIndex,
								bMethodError 		=> bMethodError,
								MethodErrorMsg 		=> MethodErrorMsg);

//Check if free space available	
	IF iDocCount >= DOC_ARRAY_SIZE OR iFreeSpaceCount = 0 THEN						//Error
		bMethodError := TRUE;		
		MethodErrorMsg.wErrorNo := GVL_DocManagement_ERROR_IDS.ERR_DOC_CAN_NOT_BE_INSERTED_THUS_ARRAY_FULL + GVL_DocManagement.wErrorIdOffset;
		
	ELSE																		//Executing, thus space available
				
			iDocIdSet := SEL(ID = 0, ID, iHighestDocID +1);						//set doc id (either defined by SPS or by host)		
					
			IF iDocIdSet <= iHighestDocId THEN										//Error, ID not higher than existing
				
				bMethodError := TRUE;
				
				//Check if ID existend already
					M_FindDoc(iDocID := ID, bDocFound => bDocIdExisting);
					
					IF bDocIdExisting THEN	//determine error details		
						MethodErrorMsg.wErrorNo := GVL_DocManagement_ERROR_IDS.ERR_DOC_CAN_NOT_BE_INSERTED_THUS_DOC_ID_EXISTENT_ALREADY + GVL_DocManagement.wErrorIdOffset;
						
					ELSE					
						MethodErrorMsg.wErrorNo := GVL_DocManagement_ERROR_IDS.ERR_DOC_ID_TO_BE_INSERTED_NOT_HIGHER_THAN_EXISTING_IDS + GVL_DocManagement.wErrorIdOffset;
						
					END_IF							
			ELSE																//ID set by host and correct			
			//Insert document	
					DocList[iLastFreeArrayIndex].ID 						:= iDocIdSet;
				
				//Parameter set by SPS				
					DocList[iLastFreeArrayIndex].Free 						:= FALSE;					
					DocList[iLastFreeArrayIndex].bLockedBySPS				:= FALSE;
					DocList[iLastFreeArrayIndex].Released					:= TRUE;
					DocList[iLastFreeArrayIndex].PositionIndex				:= eDocPositionIndex.UNDEFINED;
					
				//Parameter set by host
					DocList[iLastFreeArrayIndex].Location 					:= Location;				
					DocList[iLastFreeArrayIndex].Module 					:= Module;
					DocList[iLastFreeArrayIndex].Path 						:= Path;
					DocList[iLastFreeArrayIndex].RedAtLocation 				:= RedAtLocation;
					DocList[iLastFreeArrayIndex].RedToLocation 				:= RedToLocation;
					DocList[iLastFreeArrayIndex].bReleaseHandshakeActive	:= bReleaseHandshakeActive;
					
					bDocsInBuffer := TRUE;
			END_IF
END_IF
END_METHOD

METHOD M_InsertNewDoc2  // allow insertion of doc ID lower then highest existing
VAR_INPUT
	ID:				UDINT;
	Module:			UINT;
	Location:		UINT; 
	Path:			UINT;
	RedAtLocation:	UINT;
	RedToLocation:	UINT;
	bReleaseHandshakeActive: BOOL; 
END_VAR
VAR_OUTPUT
	iDocIdSet : UDINT := 0;
	bMethodError : BOOL := FALSE;
	MethodErrorMsg : sErrorMsg;
END_VAR
VAR
	i : UINT;
	bDocIdExisting : BOOL := FALSE;
	
	iDocCount,
	iFreeSpaceCount :	UINT := 0;

	iLastFreeArrayIndex :	UINT := 0;	
	iSmallestDocId,
	iHighestDocId :		UDINT := 0;
END_VAR
(*
V1.0 Koster Daniel
		- initial version
V1.1 Walther Ronny, 26.01.16 complete rework:
		- sErrorMsg integrated
		- unique Error IDs added
		- setting Done, Error flag in mother FB removed
		- error checks modified, added
		- ID = 0 forces SPS to define a DocID
V1.2	Walther Ronny, 29.01.16
		-standard released value changed to TRUE
*)
MethodErrorMsg.wComponent 		:= GVL_DocManagement.wCompId;
MethodErrorMsg.sFunctionName 	:= 'M_InsertNewDoc';
MethodErrorMsg.wErrorNo 		:= GVL.ERR_NO_ERROR;

//Gather actual information
	M_GetDocArrayInformation(	iDocCount 			=> iDocCount,
								iFreeSpaceCount 	=> iFreeSpaceCount,
								iSmallestDocId 		=> iSmallestDocId,
								iHighestDocId 		=> iHighestDocId,
								iLastFreeArrayIndex => iLastFreeArrayIndex,
								bMethodError 		=> bMethodError,
								MethodErrorMsg 		=> MethodErrorMsg);

//Check if free space available	
	IF iDocCount >= DOC_ARRAY_SIZE OR iFreeSpaceCount = 0 THEN						//Error
		bMethodError := TRUE;		
		MethodErrorMsg.wErrorNo := GVL_DocManagement_ERROR_IDS.ERR_DOC_CAN_NOT_BE_INSERTED_THUS_ARRAY_FULL + GVL_DocManagement.wErrorIdOffset;
		
	ELSE																		//Executing, thus space available
				
			iDocIdSet := SEL(ID = 0, ID, iHighestDocID +1);						//set doc id (either defined by SPS or by host)		
					
			IF iDocIdSet <= iHighestDocId THEN									//if ID higher than existing, check if ID exist
				
				//Check if ID existend already
					M_FindDoc(iDocID := ID, bDocFound => bDocIdExisting);
			
					IF bDocIdExisting THEN	//determine error details		
						MethodErrorMsg.wErrorNo := GVL_DocManagement_ERROR_IDS.ERR_DOC_CAN_NOT_BE_INSERTED_THUS_DOC_ID_EXISTENT_ALREADY + GVL_DocManagement.wErrorIdOffset;
						bMethodError := TRUE;
					END_IF	
			
			END_IF	
											
			IF NOT bMethodError THEN														//ID set by host and correct			
			//Insert document	
					DocList[iLastFreeArrayIndex].ID 						:= iDocIdSet;
				
				//Parameter set by SPS				
					DocList[iLastFreeArrayIndex].Free 						:= FALSE;					
					DocList[iLastFreeArrayIndex].bLockedBySPS				:= FALSE;
					DocList[iLastFreeArrayIndex].Released					:= TRUE;
					DocList[iLastFreeArrayIndex].PositionIndex				:= eDocPositionIndex.UNDEFINED;
					
				//Parameter set by host
					DocList[iLastFreeArrayIndex].Location 					:= Location;				
					DocList[iLastFreeArrayIndex].Module 					:= Module;
					DocList[iLastFreeArrayIndex].Path 						:= Path;
					DocList[iLastFreeArrayIndex].RedAtLocation 				:= RedAtLocation;
					DocList[iLastFreeArrayIndex].RedToLocation 				:= RedToLocation;
					DocList[iLastFreeArrayIndex].bReleaseHandshakeActive	:= bReleaseHandshakeActive;
					
					bDocsInBuffer := TRUE;
			END_IF
END_IF
END_METHOD

METHOD M_RedirectDoc : BOOL
VAR_INPUT
	ID:					UDINT;
	RedAtLocation:		UINT;
	RedToLocation:		UINT;
END_VAR
VAR_OUTPUT
	bDocIdFound : 		BOOL := FALSE;
	bMethodError : 		BOOL := FALSE;
	MethodErrorMsg : 	sErrorMsg;
END_VAR
VAR
	pDoc : POINTER TO sDocument;
END_VAR
(*
V1.0 Koster Daniel
		- initial version
V1.1 Walther Ronny, 27.01.16 major rework:
		- sErrorMsg integrated
		- unique Error IDs added
		- M_FindDoc method call instead for..do
*)
MethodErrorMsg.wComponent 		:= GVL_DocManagement.wCompId;
MethodErrorMsg.sFunctionName 	:= 'M_RedirectDoc';
MethodErrorMsg.wErrorNo 		:= GVL.ERR_NO_ERROR;

//just check if doc id exists
	M_FindDoc(iDocId := ID, bDocFound => bDocIdFound, pDoc => pDoc, bMethodError => bMethodError, MethodErrorMsg => MethodErrorMsg);

IF NOT bMethodError THEN //no error	
	IF bDocIdFound THEN
		pDoc^.RedAtLocation := RedAtLocation;
		pDoc^.RedToLocation := RedToLocation;
		
	ELSE
		bMethodError 			:= TRUE;
		MethodErrorMsg.wErrorNo := GVL_DocManagement_ERROR_IDS.ERR_DOC_ID_DOES_NOT_EXIST + GVL_DocManagement.wErrorIdOffset;
		
	END_IF
	
END_IF

M_RedirectDoc := bDocIdFound;
END_METHOD

METHOD M_RemoveAllDocs : BOOL
VAR_OUTPUT
	iLockedDocs : uint := 0 ;
	bMethodError : 		BOOL := FALSE;
	MethodErrorMsg : 	sErrorMsg;
END_VAR
VAR
	i : 		UINT := 0;
END_VAR
(*
V1.0 Koster Daniel
		- initial version
V1.1 Walther Ronny, 27.01.16 major rework:
		- EmptyDoc defined, sps lock integrated
*)
MethodErrorMsg.wComponent 		:= GVL_DocManagement.wCompId;
MethodErrorMsg.sFunctionName 	:= 'M_RemoveAllDocs';
MethodErrorMsg.wErrorNo 		:= GVL.ERR_NO_ERROR;


FOR i := 0 TO (DOC_ARRAY_SIZE - 1) DO
	IF DocList[i].bLockedBySps THEN
		iLockedDocs 			:= iLockedDocs + 1;
		bMethodError 			:= TRUE;
		MethodErrorMsg.wErrorNo := GVL_DocManagement_ERROR_IDS.ERR_NOT_ALL_DOCS_COULD_BE_REMOVED_THUS_LOCKED_BY_SPS + GVL_DocManagement.wErrorIdOffset;
		
	ELSE
		DocList[i] := EMPTY_DOC;
	END_IF
END_FOR

M_RemoveAllDocs := bMethodError;

bDocsInBuffer := FALSE;
END_METHOD

METHOD M_RemoveDoc : BOOL
VAR_INPUT
	ID:			UDINT;
END_VAR
VAR_OUTPUT
	bDocIdFound : 		BOOL := FALSE;
	bMethodError : 		BOOL := FALSE;
	MethodErrorMsg : 	sErrorMsg;
END_VAR
VAR
	pDoc : POINTER TO sDocument;
END_VAR
(*
V1.0 Koster Daniel
		- initial version
V1.1 Walther Ronny, 27.01.16 major rework:
		- sErrorMsg integrated
		- unique Error IDs added
		- M_FindDoc method call instead for..do
		- EmptyDoc defined
*)
MethodErrorMsg.wComponent 		:= GVL_DocManagement.wCompId;
MethodErrorMsg.sFunctionName 	:= 'M_RemoveDoc';
MethodErrorMsg.wErrorNo 		:= GVL.ERR_NO_ERROR;


//just check if doc id exists
	M_FindDoc(iDocId := ID, bDocFound => bDocIdFound, pDoc => pDoc, bMethodError => bMethodError, MethodErrorMsg => MethodErrorMsg);

IF NOT bMethodError THEN //no error	
	IF bDocIdFound THEN
		
		IF pDoc^.bLockedBySps THEN
			bMethodError 			:= TRUE;
			MethodErrorMsg.wErrorNo := GVL_DocManagement_ERROR_IDS.ERR_DOC_CAN_NOT_BE_REMOVED_THUS_LOCKED_BY_SPS + GVL_DocManagement.wErrorIdOffset;
		
		ELSE
			pDoc^ := EMPTY_DOC;
			
		END_IF
	ELSE
		bMethodError 			:= TRUE;
		MethodErrorMsg.wErrorNo := GVL_DocManagement_ERROR_IDS.ERR_DOC_ID_DOES_NOT_EXIST + GVL_DocManagement.wErrorIdOffset;
		
	END_IF
	
END_IF

M_RemoveDoc := bDocIdFound;		//If ID is found --> return TRUE
END_METHOD

METHOD PUBLIC M_ResetDocMng
VAR
	i : UINT;
END_VAR
FOR i := 0 TO (DOC_ARRAY_SIZE - 1) DO
		DocList[i] := EMPTY_DOC;

END_FOR
END_METHOD

METHOD M_SethPath : BOOL
VAR_INPUT
	ID:			UDINT;
	Path:		UINT;
END_VAR
VAR_OUTPUT
	bDocIdFound : 		BOOL := FALSE;
	bMethodError : 		BOOL := FALSE;
	MethodErrorMsg : 	sErrorMsg;
END_VAR
VAR
	pDoc : POINTER TO sDocument;
END_VAR
(*
V1.0 Koster Daniel
		- initial version
V1.1 Walther Ronny, 27.01.16 major rework:
		- sErrorMsg integrated
		- unique Error IDs added
		- M_FindDoc method call instead for..do
*)
MethodErrorMsg.wComponent 		:= GVL_DocManagement.wCompId;
MethodErrorMsg.sFunctionName 	:= 'M_SethPath';
MethodErrorMsg.wErrorNo 		:= GVL.ERR_NO_ERROR;

//just check if doc id exists
	M_FindDoc(iDocId := ID, bDocFound => bDocIdFound, pDoc => pDoc, bMethodError => bMethodError, MethodErrorMsg => MethodErrorMsg);

IF NOT bMethodError THEN //no error	
	IF bDocIdFound THEN
		pDoc^.Path := Path;
		
	ELSE
		bMethodError 			:= TRUE;
		MethodErrorMsg.wErrorNo := GVL_DocManagement_ERROR_IDS.ERR_DOC_ID_DOES_NOT_EXIST + GVL_DocManagement.wErrorIdOffset;
		
	END_IF
	
END_IF

M_SethPath := bDocIdFound;
END_METHOD

METHOD M_SetReleased : BOOL
VAR_INPUT
	ID:			UDINT;
END_VAR
VAR_OUTPUT
	bDocIdFound : 		BOOL := FALSE;
	bMethodError : 		BOOL := FALSE;
	MethodErrorMsg : 	sErrorMsg;
END_VAR
VAR
	pDoc : POINTER TO sDocument;
END_VAR
(*
V1.0 Koster Daniel
		- initial version
V1.1 Walther Ronny, 27.01.16 major rework:
		- sErrorMsg integrated
		- unique Error IDs added
		- M_FindDoc method call instead for..do
		- sps lock
*)
MethodErrorMsg.wComponent 		:= GVL_DocManagement.wCompId;
MethodErrorMsg.sFunctionName 	:= 'M_SetReleased';
MethodErrorMsg.wErrorNo 		:= GVL.ERR_NO_ERROR;

//just check if doc id exists
	M_FindDoc(iDocId := ID, bDocFound => bDocIdFound, pDoc => pDoc, bMethodError => bMethodError, MethodErrorMsg => MethodErrorMsg);

IF NOT bMethodError THEN //no error	
	IF bDocIdFound THEN
		IF pDoc^.Released = FALSE THEN
			pDoc^.Released := TRUE;
			
		ELSE
			bMethodError 			:= TRUE;
			MethodErrorMsg.wErrorNo := GVL_DocManagement_ERROR_IDS.ERR_DOC_CAN_NOT_BE_RELEASED_THUS_NOT_UNRELEASED  + GVL_DocManagement.wErrorIdOffset;	
			
		END_IF
		
	ELSE
		bMethodError 			:= TRUE;
		MethodErrorMsg.wErrorNo := GVL_DocManagement_ERROR_IDS.ERR_DOC_ID_DOES_NOT_EXIST + GVL_DocManagement.wErrorIdOffset;
		
	END_IF
	
END_IF
M_SetReleased := bMethodError;
END_METHOD

PROPERTY PUBLIC P_iArraySize : uint
GET
P_iArraySize := DOC_ARRAY_SIZE;
END_GET
END_PROPERTY

END_PROGRAM

// DocManagement/DocManagement_Ext
//Author: 				Walther Ronny
//Version:				1.0
//Last change:			14.04.16
//See Release notes at the bottom

PROGRAM DocManagement_Ext
VAR CONSTANT
	DOC_ARRAY_SIZE				:			UINT:= 500; //{warning 'RON - doc array temporarly huge!'}								
	EMPTY_DOCUMENT_PROCESSING 	: ST_Document_Processing 	:= (								
									Released 				:= TRUE,
									bReleaseHandshakeActive := TRUE,
									bLockedBySps 			:= FALSE,
									Error 					:= FALSE
									);
	EMPTY_DOC 					: ST_Document 				:= (
									Free 					:= TRUE, 
									stProcessing 			:= EMPTY_DOCUMENT_PROCESSING	
									);
END_VAR
VAR
	DocList:			ARRAY[0..(DOC_ARRAY_SIZE-1)] OF ST_Document;
END_VAR
VAR_OUTPUT
	bDocsInBuffer: BOOL;
END_VAR

(*
V1.0 Ronny Walther 28.07.17
		- initial version extended with ST_ErrorMsg and modified ST_Document struct
*)

METHOD PUBLIC M_CheckDocsInPrevLocation
VAR_INPUT
	iCurLocation : UINT;
END_VAR
VAR_OUTPUT
	iDocsInPreviousLocation : UINT := 0;
	iSmallestID : UDINT;
END_VAR
VAR
	i:UINT;
END_VAR
(*
V1.0  Walther Ronny, 23.12.15
		- initial version
*)
iSmallestID := 16#FFFF;	
		
		//Count docs in previous location and find their smallest ID
		FOR i := 0 TO (DOC_ARRAY_SIZE - 1) DO
		
			IF NOT DocList[i].Free AND DocList[i].stPosition.Location = iCurLocation-1 THEN
				
				iDocsInPreviousLocation := iDocsInPreviousLocation + 1;
				
				IF iSmallestID > DocList[i].ID THEN
					iSmallestID := DocList[i].ID;
				END_IF
			END_IF
	
		END_FOR
END_METHOD

METHOD public M_FindDoc
VAR_INPUT
	iDocID : UDINT;
END_VAR
VAR_OUTPUT
	bDocFound : 		BOOL := FALSE;
	pDoc : 				POINTER TO ST_Document; //pointer to found document
	bMethodError : 		BOOL := FALSE;
	MethodErrorMsg : 	ST_ErrorMsg;
END_VAR
VAR
	i : UINT;
END_VAR
(*
V1.0  Walther Ronny, 23.12.15
		- initial version, check if free
*)
MethodErrorMsg.wComponent 		:= GVL_DocManagement.wCompId;
MethodErrorMsg.sFunctionName 	:= 'M_GetDocInfoById';
MethodErrorMsg.wErrorNo 		:= GVL.ERR_NO_ERROR;

IF iDocID = 0 THEN
	bMethodError 				:= TRUE;			
	MethodErrorMsg.wErrorNo 	:= GVL_DocManagement_ERROR_IDS.ERR_DOC_ID_ZERO_INVALID + GVL_DocManagement.wErrorIdOffset;
	
ELSE
	//Find doc
	 FOR i := 0 TO (DOC_ARRAY_SIZE - 1) DO
					
		IF DocList[i].ID = iDocID AND NOT bDocFound AND NOT DocList[i].Free THEN
			pDoc := ADR(DocList[i]);
			bDocFound := TRUE;
			
		END_IF
					
	END_FOR
END_IF
END_METHOD

METHOD PUBLIC M_GetDocArrayInformation
VAR_OUTPUT
	iDocCount,
	iNumOfLockedDocs,
	iNumOfUnReleasedDocs,
	iNumOfDocsInLocationZero,
	iFreeSpaceCount :		UINT := 0;
		
	iSmallestDocId,
	iHighestDocId :			UDINT := 0;
	
	iLastFreeArrayIndex	 :	UINT := 0;
	
	bMethodError : 			BOOL := FALSE;
	MethodErrorMsg : 		ST_ErrorMsg;
END_VAR
VAR
	i : UINT;
END_VAR
(*
V1.0  Walther Ronny, 27.12.15
		- initial version
*)
MethodErrorMsg.wComponent 		:= GVL_DocManagement.wCompId;
MethodErrorMsg.sFunctionName 	:= 'M_GetDocArrayInformation';
MethodErrorMsg.wErrorNo 		:= GVL.ERR_NO_ERROR;

	//Find doc
	 FOR i := 0 TO (DOC_ARRAY_SIZE - 1) DO
		
		IF DocList[i].Free THEN
			//Determine free spaces
		 		iFreeSpaceCount := iFreeSpaceCount +1;
				
			//Determine last free array index
				iLastFreeArrayIndex := i;
		ELSE
			//Count docs
				iDocCount := iDocCount + 1;
				
			//Determine highest ID
				IF DocList[i].ID >	iHighestDocId THEN
					iHighestDocId := DocList[i].ID;
				END_IF
			
			//Determine smallest ID	
				IF DocList[i].ID < iSmallestDocId OR iSmallestDocId = 0 THEN
					iSmallestDocId := DocList[i].ID;
				END_IF
				
			//Determine Num of locked docs
				IF DocList[i].stProcessing.bLockedBySps THEN
					iNumOfLockedDocs := iNumOfLockedDocs + 1;
				END_IF
				
			//Determine Num of unreleased docs
				IF NOT DocList[i].stProcessing.Released THEN
					iNumOfUnReleasedDocs := iNumOfUnReleasedDocs + 1;
				END_IF
				
			//Determine Num of docs in location 0 (=buffer and ready to be processed)
				IF DocList[i].stPosition.Location = 0 THEN
					iNumOfDocsInLocationZero := iNumOfDocsInLocationZero + 1;
				END_IF
				
				
		END_IF
			

					
	END_FOR
END_METHOD

METHOD M_GetDocInfoById : ST_Document
VAR_INPUT
	ID:			UDINT;
END_VAR
VAR_OUTPUT
	bDocFound : 		BOOL := FALSE;
	bMethodError : 		BOOL := FALSE;
	MethodErrorMsg : 	ST_ErrorMsg;
END_VAR
VAR
	i : 				UINT;
	pDoc : 				POINTER TO ST_Document;
	FoundDoc : 			ST_Document;
	bDocIdFound : 		BOOL := FALSE;
END_VAR
(*
V1.0 Koster Daniel
		- initial version
V1.1 Walther Ronny, 26.01.16 major rework:
		- sErrorMsg integrated
		- unique Error IDs added
		- setting Done, Error flag in mother FB removed
		- no error, if not found but result flag
*)
MethodErrorMsg.wComponent 		:= GVL_DocManagement.wCompId;
MethodErrorMsg.sFunctionName 	:= 'M_GetDocInfoById';
MethodErrorMsg.wErrorNo 		:= GVL.ERR_NO_ERROR;

//just check if doc id exists
	M_FindDoc(iDocId := ID, bDocFound => bDocFound, pDoc => pDoc, bMethodError => bMethodError, MethodErrorMsg => MethodErrorMsg);
	
IF NOT bMethodError THEN
	IF bDocFound THEN
		FoundDoc := pDoc^;	//Document found 	
	
	ELSE
		bMethodError := TRUE;		
		MethodErrorMsg.wErrorNo := GVL_DocManagement_ERROR_IDS.ERR_DOC_ID_DOES_NOT_EXIST + GVL_DocManagement.wErrorIdOffset;
	
	END_IF
END_IF
M_GetDocInfoById := FoundDoc;
END_METHOD

METHOD PUBLIC M_Initialize
VAR_INPUT
	wCompId 			: tErrorConstant;		//TRUE => Logging activated, FALSE => Logging deactivated
	wErrorIdOffset		: tErrorConstant;		//Offset to be added to all ErrorId´s

END_VAR
GVL_DocManagement.wCompId 			:= wCompId;
GVL_DocManagement.wErrorIdOffset 	:= wErrorIdOffset;
END_METHOD

METHOD M_InsertNewDoc
VAR_INPUT
	ID:				UDINT;
	Module:			UINT;
	Location:		UINT; 
	Path:			UINT;
	RedAtLocation:	UINT;
	RedToLocation:	UINT;
	bReleaseHandshakeActive: BOOL; 
	DataString : STRING(GVL_DocManagement.MAX_INFO_TEXT_SIZE);
	DataField1 : LREAL;
	DataField2 : UDINT;
	DataField3 : UINT;
	DataField4 : BYTE;
END_VAR
VAR_OUTPUT
	iDocIdSet : UDINT := 0;
	bMethodError : BOOL := FALSE;
	MethodErrorMsg : ST_ErrorMsg;
END_VAR
VAR
	i : UINT;
	bDocIdExisting : BOOL := FALSE;
	
	iDocCount,
	iFreeSpaceCount :	UINT := 0;

	iLastFreeArrayIndex :	UINT := 0;	
	iSmallestDocId,
	iHighestDocId :		UDINT := 0;
END_VAR
(*
V1.0 Koster Daniel
		- initial version
V1.1 Walther Ronny, 26.01.16 complete rework:
		- sErrorMsg integrated
		- unique Error IDs added
		- setting Done, Error flag in mother FB removed
		- error checks modified, added
		- ID = 0 forces SPS to define a DocID
V1.2	Walther Ronny, 29.01.16
		-standard released value changed to TRUE
*)
MethodErrorMsg.wComponent 		:= GVL_DocManagement.wCompId;
MethodErrorMsg.sFunctionName 	:= 'M_InsertNewDoc';
MethodErrorMsg.wErrorNo 		:= GVL.ERR_NO_ERROR;

//Gather actual information
	M_GetDocArrayInformation(	iDocCount 			=> iDocCount,
								iFreeSpaceCount 	=> iFreeSpaceCount,
								iSmallestDocId 		=> iSmallestDocId,
								iHighestDocId 		=> iHighestDocId,
								iLastFreeArrayIndex => iLastFreeArrayIndex,
								bMethodError 		=> bMethodError,
								MethodErrorMsg 		=> MethodErrorMsg);

//Check if free space available	
	IF iDocCount >= DOC_ARRAY_SIZE OR iFreeSpaceCount = 0 THEN						//Error
		bMethodError := TRUE;		
		MethodErrorMsg.wErrorNo := GVL_DocManagement_ERROR_IDS.ERR_DOC_CAN_NOT_BE_INSERTED_THUS_ARRAY_FULL + GVL_DocManagement.wErrorIdOffset;
		
	ELSE																		//Executing, thus space available
			
			iDocIdSet := SEL(ID = 0, ID, iHighestDocID +1);						//set doc id (either defined by SPS or by host)				
									
			IF iDocIdSet <= iHighestDocId THEN											//Error, ID not higher than existing
				
				bMethodError := TRUE;
				
				//Check if ID existend already
					M_FindDoc(iDocID := ID, bDocFound => bDocIdExisting);
					
					IF bDocIdExisting THEN	//determine error details		
						MethodErrorMsg.wErrorNo := GVL_DocManagement_ERROR_IDS.ERR_DOC_CAN_NOT_BE_INSERTED_THUS_DOC_ID_EXISTENT_ALREADY + GVL_DocManagement.wErrorIdOffset;
						
					ELSE					
						MethodErrorMsg.wErrorNo := GVL_DocManagement_ERROR_IDS.ERR_DOC_ID_TO_BE_INSERTED_NOT_HIGHER_THAN_EXISTING_IDS + GVL_DocManagement.wErrorIdOffset;
						
					END_IF
							
			ELSE																//ID set by host and correct
							//Insert document	
					DocList[iLastFreeArrayIndex].ID 									:= iDocIdSet;
				
				//Parameter set by SPS				
					DocList[iLastFreeArrayIndex].Free 									:= FALSE;					
					DocList[iLastFreeArrayIndex].stProcessing.bLockedBySPS				:= FALSE;
					DocList[iLastFreeArrayIndex].stProcessing.Released					:= TRUE;
					
				//Parameter set by host
					DocList[iLastFreeArrayIndex].stPosition.Location 					:= Location;				
					DocList[iLastFreeArrayIndex].stPosition.Module 						:= Module;
					DocList[iLastFreeArrayIndex].stPath.Path 							:= Path;
					DocList[iLastFreeArrayIndex].stPath.RedAtLocation 					:= RedAtLocation;
					DocList[iLastFreeArrayIndex].stPath.RedToLocation 					:= RedToLocation;
					DocList[iLastFreeArrayIndex].stProcessing.bReleaseHandshakeActive	:= bReleaseHandshakeActive;
					
					DocList[iLastFreeArrayIndex].stAdditionalData.DataString			:= DataString;
					DocList[iLastFreeArrayIndex].stAdditionalData.DataField1			:= DataField1;
					DocList[iLastFreeArrayIndex].stAdditionalData.DataFiled2			:= DataField2;
					DocList[iLastFreeArrayIndex].stAdditionalData.DataField3			:= DataField3;
					DocList[iLastFreeArrayIndex].stAdditionalData.DataField4			:= DataField4;
					
					bDocsInBuffer := TRUE;
			END_IF			
END_IF
END_METHOD

METHOD M_RedirectDoc : BOOL
VAR_INPUT
	ID:					UDINT;
	RedAtLocation:		UINT;
	RedToLocation:		UINT;
END_VAR
VAR_OUTPUT
	bDocIdFound : 		BOOL := FALSE;
	bMethodError : 		BOOL := FALSE;
	MethodErrorMsg : 	ST_ErrorMsg;
END_VAR
VAR
	pDoc : POINTER TO ST_Document;
END_VAR
(*
V1.0 Koster Daniel
		- initial version
V1.1 Walther Ronny, 27.01.16 major rework:
		- sErrorMsg integrated
		- unique Error IDs added
		- M_FindDoc method call instead for..do
*)
MethodErrorMsg.wComponent 		:= GVL_DocManagement.wCompId;
MethodErrorMsg.sFunctionName 	:= 'M_RedirectDoc';
MethodErrorMsg.wErrorNo 		:= GVL.ERR_NO_ERROR;

//just check if doc id exists
	M_FindDoc(iDocId := ID, bDocFound => bDocIdFound, pDoc => pDoc, bMethodError => bMethodError, MethodErrorMsg => MethodErrorMsg);

IF NOT bMethodError THEN //no error	
	IF bDocIdFound THEN
		pDoc^.stPath.RedAtLocation := RedAtLocation;
		pDoc^.stPath.RedToLocation := RedToLocation;
		
	ELSE
		bMethodError 			:= TRUE;
		MethodErrorMsg.wErrorNo := GVL_DocManagement_ERROR_IDS.ERR_DOC_ID_DOES_NOT_EXIST + GVL_DocManagement.wErrorIdOffset;
		
	END_IF
	
END_IF

M_RedirectDoc := bDocIdFound;
END_METHOD

METHOD M_RemoveAllDocs : BOOL
VAR_OUTPUT
	iLockedDocs : uint := 0 ;
	bMethodError : 		BOOL := FALSE;
	MethodErrorMsg : 	ST_ErrorMsg;
END_VAR
VAR
	i : 		UINT := 0;
END_VAR
(*
V1.0 Koster Daniel
		- initial version
V1.1 Walther Ronny, 27.01.16 major rework:
		- EmptyDoc defined, sps lock integrated
*)
MethodErrorMsg.wComponent 		:= GVL_DocManagement.wCompId;
MethodErrorMsg.sFunctionName 	:= 'M_RemoveAllDocs';
MethodErrorMsg.wErrorNo 		:= GVL.ERR_NO_ERROR;


FOR i := 0 TO (DOC_ARRAY_SIZE - 1) DO
	IF DocList[i].stProcessing.bLockedBySps THEN
		iLockedDocs 			:= iLockedDocs + 1;
		bMethodError 			:= TRUE;
		MethodErrorMsg.wErrorNo := GVL_DocManagement_ERROR_IDS.ERR_NOT_ALL_DOCS_COULD_BE_REMOVED_THUS_LOCKED_BY_SPS + GVL_DocManagement.wErrorIdOffset;
		
	ELSE
		DocList[i] := EMPTY_DOC;
	END_IF
END_FOR

M_RemoveAllDocs := bMethodError;

bDocsInBuffer := FALSE;
END_METHOD

METHOD M_RemoveDoc : BOOL
VAR_INPUT
	ID:			UDINT;
END_VAR
VAR_OUTPUT
	bDocIdFound : 		BOOL := FALSE;
	bMethodError : 		BOOL := FALSE;
	MethodErrorMsg : 	ST_ErrorMsg;
END_VAR
VAR
	pDoc : POINTER TO ST_Document;
END_VAR
(*
V1.0 Koster Daniel
		- initial version
V1.1 Walther Ronny, 27.01.16 major rework:
		- sErrorMsg integrated
		- unique Error IDs added
		- M_FindDoc method call instead for..do
		- EmptyDoc defined
*)
MethodErrorMsg.wComponent 		:= GVL_DocManagement.wCompId;
MethodErrorMsg.sFunctionName 	:= 'M_RemoveDoc';
MethodErrorMsg.wErrorNo 		:= GVL.ERR_NO_ERROR;


//just check if doc id exists
	M_FindDoc(iDocId := ID, bDocFound => bDocIdFound, pDoc => pDoc, bMethodError => bMethodError, MethodErrorMsg => MethodErrorMsg);

IF NOT bMethodError THEN //no error	
	IF bDocIdFound THEN
		
		IF pDoc^.stProcessing.bLockedBySps THEN
			bMethodError 			:= TRUE;
			MethodErrorMsg.wErrorNo := GVL_DocManagement_ERROR_IDS.ERR_DOC_CAN_NOT_BE_REMOVED_THUS_LOCKED_BY_SPS + GVL_DocManagement.wErrorIdOffset;
		
		ELSE
			pDoc^ := EMPTY_DOC;
			
		END_IF
	ELSE
		bMethodError 			:= TRUE;
		MethodErrorMsg.wErrorNo := GVL_DocManagement_ERROR_IDS.ERR_DOC_ID_DOES_NOT_EXIST + GVL_DocManagement.wErrorIdOffset;
		
	END_IF
	
END_IF

M_RemoveDoc := bDocIdFound;		//If ID is found --> return TRUE
END_METHOD

METHOD PUBLIC M_ResetDocMng
VAR
	i : UINT;
END_VAR
FOR i := 0 TO (DOC_ARRAY_SIZE - 1) DO
		DocList[i] := EMPTY_DOC;

END_FOR
END_METHOD

METHOD M_SethPath : BOOL
VAR_INPUT
	ID:			UDINT;
	Path:		UINT;
END_VAR
VAR_OUTPUT
	bDocIdFound : 		BOOL := FALSE;
	bMethodError : 		BOOL := FALSE;
	MethodErrorMsg : 	ST_ErrorMsg;
END_VAR
VAR
	pDoc : POINTER TO ST_Document;
END_VAR
(*
V1.0 Koster Daniel
		- initial version
V1.1 Walther Ronny, 27.01.16 major rework:
		- sErrorMsg integrated
		- unique Error IDs added
		- M_FindDoc method call instead for..do
*)
MethodErrorMsg.wComponent 		:= GVL_DocManagement.wCompId;
MethodErrorMsg.sFunctionName 	:= 'M_SethPath';
MethodErrorMsg.wErrorNo 		:= GVL.ERR_NO_ERROR;

//just check if doc id exists
	M_FindDoc(iDocId := ID, bDocFound => bDocIdFound, pDoc => pDoc, bMethodError => bMethodError, MethodErrorMsg => MethodErrorMsg);

IF NOT bMethodError THEN //no error	
	IF bDocIdFound THEN
		pDoc^.stPath.Path := Path;
		
	ELSE
		bMethodError 			:= TRUE;
		MethodErrorMsg.wErrorNo := GVL_DocManagement_ERROR_IDS.ERR_DOC_ID_DOES_NOT_EXIST + GVL_DocManagement.wErrorIdOffset;
		
	END_IF
	
END_IF

M_SethPath := bDocIdFound;
END_METHOD

METHOD M_SetReleased : BOOL
VAR_INPUT
	ID:			UDINT;
END_VAR
VAR_OUTPUT
	bDocIdFound : 		BOOL := FALSE;
	bMethodError : 		BOOL := FALSE;
	MethodErrorMsg : 	ST_ErrorMsg;
END_VAR
VAR
	pDoc : POINTER TO ST_Document;
END_VAR
(*
V1.0 Koster Daniel
		- initial version
V1.1 Walther Ronny, 27.01.16 major rework:
		- sErrorMsg integrated
		- unique Error IDs added
		- M_FindDoc method call instead for..do
		- sps lock
*)
MethodErrorMsg.wComponent 		:= GVL_DocManagement.wCompId;
MethodErrorMsg.sFunctionName 	:= 'M_SetReleased';
MethodErrorMsg.wErrorNo 		:= GVL.ERR_NO_ERROR;

//just check if doc id exists
	M_FindDoc(iDocId := ID, bDocFound => bDocIdFound, pDoc => pDoc, bMethodError => bMethodError, MethodErrorMsg => MethodErrorMsg);

IF NOT bMethodError THEN //no error	
	IF bDocIdFound THEN
		IF pDoc^.stProcessing.Released = FALSE THEN
			pDoc^.stProcessing.Released := TRUE;
			
		ELSE
			bMethodError 			:= TRUE;
			MethodErrorMsg.wErrorNo := GVL_DocManagement_ERROR_IDS.ERR_DOC_CAN_NOT_BE_RELEASED_THUS_NOT_UNRELEASED  + GVL_DocManagement.wErrorIdOffset;	
			
		END_IF
		
	ELSE
		bMethodError 			:= TRUE;
		MethodErrorMsg.wErrorNo := GVL_DocManagement_ERROR_IDS.ERR_DOC_ID_DOES_NOT_EXIST + GVL_DocManagement.wErrorIdOffset;
		
	END_IF
	
END_IF
M_SetReleased := bMethodError;
END_METHOD

PROPERTY PUBLIC P_iArraySize : uint
GET
P_iArraySize := DOC_ARRAY_SIZE;
END_GET
END_PROPERTY

END_PROGRAM

// ErrorManagement/ErrorManagement_Ext
//Author: 				Koster Daniel, Walther Ronny
//Version:				1.0
//Last change:			24.07.17
//See Release notes at the bottom
PROGRAM ErrorManagement_Ext
VAR
	pErrHnd : POINTER TO FB_ErrorHandler_Base;
	
	iSysErrorMsgIdCounter :		UINT := 1;		//Counter to create unique ErrorMsg ID
	SysErrorList:				ARRAY[0..(ERROR_ARRAY_SIZE-1)] OF ST_SystemError;
	

	//Automatic periodical Event sending
		tEventIntervalTime : 		TIME := ERROR_EVENT_SENDING_CYCLE_TIME;
		tEventIntervalTimer :		TON;
		iEvtSendingIndex :			UINT := 0;	//Index while scrolling thru error list inside M_SendEvents method
	
	//Event sending mode flags	
		CurNotificationMode : 			eErrorNotificationMode := ERROR_NOTIFICATION_MODE;
		
		bEventSendingOnceActive : 		BOOL := FALSE;	

//Note: The following objects are used like constants, but thus wComponent is set first when the program is initialized they can not be declared as constants!
	NULL_ERROR_MSG : 	ST_ErrorMsg 		:= (	wModule 		:= 1,
												pErrorHandler 	:= ADR(ErrHand_Dummy),
												wComponent 		:= GVL_ErrorManagement.wCompId,
												sFunctionName 	:= '***NULL_ERROR***',
												eErrorLevel		:= E_ErrorLevels._ERROR,
												wErrorNo 		:= GVL.ERR_NO_ERROR);	
	
	NULL_ERROR : 		ST_SystemError 	:= (	SysErrorMessageID 	:= 0,
												ErrorMsg 			:= NULL_ERROR_MSG);	
	ErrHand_Dummy :		FB_ErrorHandler_Base();	
END_VAR
VAR CONSTANT
	ERROR_ARRAY_SIZE:					UINT:= 40;			//size of error array
	ERROR_NOTIFICATION_MODE :			UINT := eErrorNotificationMode.SENDING_ERRORS_ONCE_IMMEDIATLY;
	ERROR_EVENT_SENDING_CYCLE_TIME : 	TIME := T#200MS;	//periodic event sending intervall
	

								
	EMPTY_SYS_ERROR : 	ST_SystemError 	:= (	SysErrorMessageID 	:= 0);	
	

END_VAR
(*
V1.0 Walther Ronny, 24.07.16:
	- extension of original Errormanagement.prg
	- 2 different error events added (SPS + Twincat). 
		This means, that ErrorMsg defines if its a SPS or Twincat error and this will control to which Event variable the error is sent later on. 
		This avoids misinterpretation thus both errors use different IDs.
	- ST_ErrorMsg, E_ErrorTypes, E_ErrorLevels modified
*)

//automatic sending modes
	M_SendEvents();

METHOD PUBLIC M_GetErrorArrayInformation
VAR_OUTPUT
	iErrorCount,
	iFreeSpaceCount :		UINT := 0;	
	
	bMethodError : 			BOOL := FALSE;
	MethodErrorMsg : 		ST_ErrorMsg;
END_VAR
VAR
	i : UINT;
END_VAR
(*
V1.0  Walther Ronny, 27.12.15
		- initial version
*)
MethodErrorMsg.wComponent 		:= GVL_ErrorManagement.wCompId;
MethodErrorMsg.sFunctionName 	:= 'M_GetErrorArrayInformation';
MethodErrorMsg.wErrorNo 		:= GVL.ERR_NO_ERROR;

//scroll errors
	 FOR i := 0 TO (ERROR_ARRAY_SIZE - 1) DO
		
		IF SysErrorList[i].SysErrorMessageID = 0 THEN //0 => empty THEN
			//Determine free spaces
		 		inc(iFreeSpaceCount);
			
		ELSE
			//Count errors
				inc(iErrorCount);
				
		END_IF								
	END_FOR
END_METHOD

METHOD PUBLIC M_GetErrorInfo : ST_SystemError	//Gives back the Info for the SysError with ErrorID = ErrorID
VAR_INPUT
	iSysErrorMsgId:	UINT;
END_VAR
VAR_OUTPUT
	bErrorMsgIdFound : 	BOOL := FALSE;
	bMethodError : 		BOOL := FALSE;
	MethodErrorMsg : 	ST_ErrorMsg;
END_VAR
VAR 
	i : UINT;
END_VAR
MethodErrorMsg.wComponent 		:= GVL_ErrorManagement.wCompId;
MethodErrorMsg.sFunctionName 	:= 'M_GetErrorInfo';
MethodErrorMsg.wErrorNo 		:= GVL.ERR_NO_ERROR;

IF iSysErrorMsgId = 0 THEN		
	bMethodError := TRUE;
	MethodErrorMsg.wErrorNo := GVL_ErrorManagement_ERROR_IDS.ERR_ERROR_ID_ZERO_INVALID + GVL_ErrorManagement.wErrorIdOffset;
	
ELSE
	FOR i := 0 TO (ERROR_ARRAY_SIZE - 1) DO
		IF SysErrorList[i].SysErrorMessageID = iSysErrorMsgId THEN	//ErrorID is found
			bErrorMsgIdFound := TRUE;			
			
			M_GetErrorInfo := SysErrorList[i];
			EXIT;			
		END_IF
	END_FOR
END_IF

IF NOT bErrorMsgIdFound THEN//If ErrorID couldn´t be found
	bMethodError := TRUE;
	MethodErrorMsg.wErrorNo := GVL_ErrorManagement_ERROR_IDS.ERR_ERROR_ID_NOT_FOUND + GVL_ErrorManagement.wErrorIdOffset;
	
END_IF
END_METHOD

METHOD PUBLIC M_Initialize
VAR_INPUT
	wCompId 			: tErrorConstant;	//TRUE => Logging activated, FALSE => Logging deactivated
	wErrorIdOffset		: tErrorConstant;	//Offset to be added to all ErrorId´s (except Twincat errors)	
	bLoggingOnOff 		: BOOL;				//TRUE => Logging activated, FALSE => Logging deactivated
	pEvt_SpsError 		: POINTER TO ST_SystemErrorEvent;
	pEvt_TwincatError 	: POINTER TO ST_SystemErrorEvent;
END_VAR
GVL_ErrorManagement.wCompId 		:= wCompId;
GVL_ErrorManagement.wErrorIdOffset 	:= wErrorIdOffset;
GVL_ErrorManagement.bLoggingOnOff	:= bLoggingOnOff;


//Check Evt pointer, if invalid set dummy
	IF IsValidPtr(pEvt_SpsError) THEN
		GVL_ErrorManagement.pEvt_SpsError 	:= pEvt_SpsError;
		
	ELSE		
		GVL_ErrorManagement.pEvt_SpsError := ADR(GVL_ErrorManagement.cDUMMY_EVENT);

	END_IF
	//Check Evt pointer, if invalid set dummy
	IF IsValidPtr(pEvt_TwincatError) THEN
		GVL_ErrorManagement.pEvt_TwincatError 	:= pEvt_TwincatError;
		
	ELSE		
		GVL_ErrorManagement.pEvt_TwincatError := ADR(GVL_ErrorManagement.cDUMMY_EVENT);

	END_IF
END_METHOD

METHOD PUBLIC M_InsertNewError		//Puts new SysError in the SysError List
VAR_INPUT
	ErrorMsg 		: ST_ErrorMsg;
END_VAR
VAR_OUTPUT
	iSysErrorMsgId : 	UINT := 0;
	bMethodError : 		BOOL := FALSE;
	MethodErrorMsg : 	ST_ErrorMsg;
END_VAR
VAR
	bErrorSet : 		BOOL := FALSE;
	i : 				UINT := 0;
END_VAR
MethodErrorMsg.wComponent 		:= GVL_ErrorManagement.wCompId;
MethodErrorMsg.sFunctionName 	:= 'M_InsertNewSysError';
MethodErrorMsg.wErrorNo 		:= GVL.ERR_NO_ERROR;


FOR i := 0 TO (ERROR_ARRAY_SIZE - 1) DO
	IF SysErrorList[i].SysErrorMessageID = 0 THEN //0 => empty
		iSysErrorMsgId := iSysErrorMsgIdCounter;
		
		SysErrorList[i].SysErrorMessageID 	:= iSysErrorMsgId;
		SysErrorList[i].ErrorMsg 			:= ErrorMsg;	
		SysErrorList[i].bErrorWasSent		:= FALSE;
		
		//Handle not set variables
			IF NOT IsValidPtr(SysErrorList[i].ErrorMsg.pErrorHandler) THEN
				SysErrorList[i].ErrorMsg.pErrorHandler := ADR(ErrHand_Dummy);
			END_IF
			IF SysErrorList[i].ErrorMsg.eErrorLevel = E_ErrorLevels._UNDEFINED THEN //otherwise 0 is always a fatal error for PIA
				 SysErrorList[i].ErrorMsg.eErrorLevel := E_ErrorLevels._ERROR;
			END_IF
		//Logging
			M_CreateLogData(pErr := SysErrorList[i]);
			
		inc(iSysErrorMsgIdCounter);
		bErrorSet := TRUE;
		
		EXIT;
	END_IF
END_FOR

IF NOT bErrorSet THEN
	MethodErrorMsg.wErrorNo 		:= GVL_ErrorManagement_ERROR_IDS.ERR_ERROR_ARRAY_FULL + GVL_ErrorManagement.wErrorIdOffset;
	bMethodError := TRUE;
END_IF
END_METHOD

METHOD PUBLIC M_RemoveAllErrors
VAR_OUTPUT
	bMethodError : 		BOOL := FALSE;
	MethodErrorMsg : 	ST_ErrorMsg;
END_VAR
VAR
	i : UINT;
	sysErr : ST_SystemError;
END_VAR
MethodErrorMsg.wComponent 		:= GVL_ErrorManagement.wCompId;
MethodErrorMsg.sFunctionName 	:= 'M_RemoveAllErrors';
MethodErrorMsg.wErrorNo 		:= GVL.ERR_NO_ERROR;


sysErr := NULL_ERROR;
sysErr.ErrorMsg.eErrorType := E_ErrorTypes.SPS;
sysErr.ErrorMsg.wComponent := GVL_ErrorManagement.wCompId;

FOR i := 0 TO (ERROR_ARRAY_SIZE - 1) DO
	SysErrorList[i] := EMPTY_SYS_ERROR;
END_FOR

//Log data	
	M_CreateLogData(pErr := sysErr);

//Create Event - NULL ERROR	
	//sps error
	M_CreateEvent(sysErr := sysErr);

	//twincat error	
	sysErr.ErrorMsg.eErrorType := E_ErrorTypes.TWINCAT;
	M_CreateEvent(sysErr := sysErr);
END_METHOD

METHOD public M_RemoveError	//Clears SysError with ErrorID = ErrorID
VAR_INPUT
	iSysErrorMsgId : 	UINT;
END_VAR
VAR_OUTPUT
	bErrorMsgIdFound : 	BOOL := FALSE;
	bMethodError : 		BOOL := FALSE;
	MethodErrorMsg : 	ST_ErrorMsg;
END_VAR
VAR
	i : UINT;
END_VAR
MethodErrorMsg.wComponent 		:= GVL_ErrorManagement.wCompId;
MethodErrorMsg.sFunctionName 	:= 'M_RemoveError';
MethodErrorMsg.wErrorNo 		:= GVL.ERR_NO_ERROR;

IF iSysErrorMsgId = 0 THEN		
	bMethodError := TRUE;
	MethodErrorMsg.wErrorNo := GVL_ErrorManagement_ERROR_IDS.ERR_ERROR_ID_ZERO_INVALID + GVL_ErrorManagement.wErrorIdOffset;
	
ELSE
	FOR i := 0 TO (ERROR_ARRAY_SIZE - 1) DO
		IF SysErrorList[i].SysErrorMessageID = iSysErrorMsgId THEN	//ErrorID is found
			bErrorMsgIdFound := TRUE;			
			
			SysErrorList[i] := EMPTY_SYS_ERROR;	//remove SysError
			EXIT;			
		END_IF
	END_FOR
END_IF

IF NOT bErrorMsgIdFound THEN//If ErrorID couldn´t be found
	bMethodError := TRUE;
	MethodErrorMsg.wErrorNo := GVL_ErrorManagement_ERROR_IDS.ERR_ERROR_ID_NOT_FOUND + GVL_ErrorManagement.wErrorIdOffset;
	
END_IF
END_METHOD

METHOD PUBLIC M_ResetSysErrorMng
M_RemoveAllErrors();
END_METHOD

METHOD PUBLIC M_SendAllErrorOnce
VAR_OUTPUT
	bMethodError : 		BOOL := FALSE;
	MethodErrorMsg : 	ST_ErrorMsg;
END_VAR
MethodErrorMsg.wComponent 		:= GVL_ErrorManagement.wCompId;
MethodErrorMsg.sFunctionName 	:= 'M_SendEvtOnce';
MethodErrorMsg.wErrorNo 		:= GVL.ERR_NO_ERROR;

IF CurNotificationMode = eErrorNotificationMode.SENDING_ERRORS_ALWAYS_PERIODICALLY THEN
	bMethodError := TRUE;
	MethodErrorMsg.wErrorNo 	:= GVL_ErrorManagement_ERROR_IDS.ERR_SEND_ERRORS_ONCE_NOT_POSSIBLE_THUS_PERIODIC_SENDING_ACTIVATED + GVL_ErrorManagement.wErrorIdOffset;
	
ELSE
	bEventSendingOnceActive := TRUE;
	
	//Reset index in order to start scanning from the beginning
		iEvtSendingIndex := 0;
END_IF
END_METHOD

METHOD PRIVATE M_SendEvents		//Sends the Event for every SysErrror in the SysError List
VAR 
	i : UINT;
	localEvt : sSystemErrorEvent;
END_VAR
//Only Intervals above 100 ms (processing cycle)
IF tEventIntervalTime < T#100MS THEN
	tEventIntervalTime := T#100MS;
END_IF

//Sending

IF tEventIntervalTimer.Q THEN
	
	tEventIntervalTimer(IN := FALSE);
	
	FOR i := iEvtSendingIndex TO (ERROR_ARRAY_SIZE-1) DO
			IF SysErrorList[i].SysErrorMessageID <> 0 THEN //not empty	
														
					IF CurNotificationMode= eErrorNotificationMode.SENDING_ERRORS_ALWAYS_PERIODICALLY OR bEventSendingOnceActive THEN	
						//send every error
						M_CreateEvent(sysErr := SysErrorList[i]);		
						SysErrorList[i].bErrorWasSent		:= TRUE;
						tEventIntervalTimer(IN := TRUE);	
					
						EXIT;
						
					ELSIF CurNotificationMode = eErrorNotificationMode.SENDING_ERRORS_ONCE_IMMEDIATLY THEN
						
						IF NOT SysErrorList[i].bErrorWasSent THEN
							//send only errors which have not been sent before
							M_CreateEvent(sysErr := SysErrorList[i]);		
							SysErrorList[i].bErrorWasSent		:= TRUE;
							tEventIntervalTimer(IN := TRUE);	
							
							EXIT;
							
						END_IF
					END_IF
					
			END_IF		
	END_FOR
		
	iEvtSendingIndex := inc(i);
	
	IF iEvtSendingIndex >= ERROR_ARRAY_SIZE THEN
		iEvtSendingIndex := 0;
		bEventSendingOnceActive := FALSE;
	END_IF
	
ELSE
	tEventIntervalTimer(IN := TRUE, PT := tEventIntervalTime);
	
END_IF
END_METHOD

METHOD PUBLIC M_SendSingleError
VAR_INPUT
	iSysErrorMsgId : UINT;
END_VAR
VAR_OUTPUT
	bErrorMsgIdFound : 	BOOL := FALSE;
	bMethodError : 		BOOL := FALSE;
	MethodErrorMsg : 	ST_ErrorMsg;
END_VAR
VAR
	sysErr : ST_SystemError;
	
END_VAR
sysErr := M_GetErrorInfo(	iSysErrorMsgID 	:= iSysErrorMsgId,
							bMethodError 	=> bMethodError,
							MethodErrorMsg 	=> MethodErrorMsg);
							
IF NOT bMethodError THEN
		M_CreateEvent(sysErr := sysErr);				
END_IF
END_METHOD

PROPERTY PUBLIC P_bHaveAllErrorsBeenSentAtLeastOnce : bool
GET
VAR
	i : UINT;
	bHaveAllBeenSend : BOOL := TRUE;;
END_VAR
FOR i := 0 TO (ERROR_ARRAY_SIZE - 1) DO
	IF SysErrorList[i].SysErrorMessageID <> 0 AND NOT SysErrorList[i].bErrorWasSent THEN
		bHaveAllBeenSend := FALSE;
		EXIT;
	END_IF
END_FOR

P_bHaveAllErrorsBeenSentAtLeastOnce := bHaveAllBeenSend;
END_GET
END_PROPERTY

PROPERTY PUBLIC P_ErrorNotificationMode : eErrorNotificationMode
GET
P_ErrorNotificationMode := CurNotificationMode;
END_GET
SET
CurNotificationMode := P_ErrorNotificationMode;
END_SET
END_PROPERTY

PROPERTY PUBLIC P_tEventIntervall : Time
GET
P_tEventIntervall := tEventIntervalTime;
END_GET
SET
tEventIntervalTime := P_tEventIntervall;
END_SET
END_PROPERTY

METHOD PRIVATE M_CreateEvent //Create an event from a system error object from array
VAR_INPUT
	sysErr : ST_SystemError;
END_VAR
VAR
	localEvt : ST_SystemErrorEvent;
END_VAR
//Prepare local evt structure				
	localEvt.SysErrorMessageID 		:= sysErr.SysErrorMessageID;
						
	localEvt.ErrorTyp 				:= sysErr.ErrorMsg.eErrorLevel;				
	localEvt.ErrorModuleId 			:= sysErr.ErrorMsg.wModule; 
	localEvt.ErrorCompId 			:= sysErr.ErrorMsg.wComponent;
	localEvt.ErrorId 				:= sysErr.ErrorMsg.wErrorNo;
	localEvt.iRelatedDocId			:= sysErr.ErrorMsg.iRelatedDocId;	
	
	IF NOT IsValidPtr(sysErr.ErrorMsg.pErrorHandler) THEN
		sysErr.ErrorMsg.pErrorHandler := ADR(ErrHand_Dummy);
		
	ELSE
		pErrHnd := sysErr.ErrorMsg.pErrorHandler;

	END_IF	 
		
	localEvt.AvailableHandlingModes := pErrHnd^.P_wAllowedHandlingModes;
	
					
//Set final evt structure
	IF sysErr.ErrorMsg.eErrorType = E_ErrorTypes.SPS THEN
		localEvt.EventChangeFlag 		:= switch(GVL_ErrorManagement.pEvt_SpsError^.EventChangeFlag);
		GVL_ErrorManagement.pEvt_SpsError^ := localEvt;
	ELSIF sysErr.ErrorMsg.eErrorType = E_ErrorTypes.TWINCAT THEN
		localEvt.EventChangeFlag 		:= switch(GVL_ErrorManagement.pEvt_TwincatError^.EventChangeFlag);
		GVL_ErrorManagement.pEvt_TwincatError^ := localEvt;
	END_IF
END_METHOD

METHOD PRIVATE M_CreateLogData
VAR_INPUT
	pErr : ST_SystemError;
END_VAR
VAR
	sFuncName: STRING;
	strModule,
	strComp,
	strErrorId,
	strRelDocId,
	strErrorTyp,
	strLogMsg : STRING;
END_VAR
IF NOT GVL_ErrorManagement.bLoggingOnOff THEN
	RETURN;
END_IF

//Create log string
	strModule := CONCAT('|Module: ',WORD_TO_STRING(pErr.ErrorMsg.wModule));
	strLogMsg := CONCAT(strLogMsg, strModule);
	
	strComp := concat('|Component: ', WORD_TO_STRING(pErr.ErrorMsg.wComponent));
	strLogMsg := CONCAT(strLogMsg, strComp);
	
	strErrorId := concat('|ErrorId: ', WORD_TO_STRING(pErr.ErrorMsg.wErrorNo));
	strLogMsg := CONCAT(strLogMsg, strErrorId);
	
	strRelDocId := concat('|RelatedDocId: ', UDINT_TO_STRING(pErr.ErrorMsg.iRelatedDocId));
	strLogMsg := CONCAT(strLogMsg, strRelDocId);
	
	strErrorTyp := concat('|ErrorTyp: ', UINT_TO_STRING(pErr.ErrorMsg.eErrorLevel));
	strLogMsg := CONCAT(strLogMsg, strErrorTyp);

	sFuncName := pErr.ErrorMsg.sFunctionName;
	
//log data
CASE pErr.ErrorMsg.eErrorLevel OF
E_ErrorLevels._ERROR : 
						Logging.Error(Caller 	:= sFuncName, 
										Msg 	:= strLogMsg);	
										
E_ErrorLevels._FATAL : 
						Logging.Fatal(Caller 	:= sFuncName, 
										Msg 	:= strLogMsg);	
										
E_ErrorLevels._WARNING : 
						Logging.Warn(	Caller 	:= sFuncName, 
										Msg 	:= strLogMsg);	
ELSE
						Logging.Trace(Caller 	:= sFuncName, 
										Msg 	:= strLogMsg);	
END_CASE
END_METHOD

END_PROGRAM

// Standard/FB_MethodState
//Author: 				Walther Ronny
//Version:				1.0
//Last change:			16.03.16
//See Release notes at the bottom
//{attribute 'hide_all_locals'}
FUNCTION_BLOCK PUBLIC FB_MethodState IMPLEMENTS ITF_MethodState //Fb to help realizing a state machine inside a method
VAR_INPUT
	tTimeout : TIME;
END_VAR
VAR
	m_CurMethodStates : sMethodState;
	m_tTimeoutTimer : TON;
END_VAR
{library PUBLIC}
VAR CONSTANT
	RESET_STATE : UINT := 0;
	START_STATE : UINT := 1;
	DONE_STATE : UINT := 99;
END_VAR
(*
V1.0 Walther Ronny
	- initial version
*)

m_tTimeoutTimer(PT:=tTimeout);

 IF 		m_tTimeoutTimer.Q 				//Timer eleapsed
	AND 	tTimeout <> T#0S 				//Ignore, if Timeout deactivated
	AND NOT m_CurMethodStates.bDone THEN	//Ignore, if Done set already
	
	 m_CurMethodStates.bError := TRUE;
	 GoDoneState();
	 
 END_IF

PROPERTY bBusy : BOOL
GET
bBusy := m_CurMethodStates.bBusy;
END_GET
END_PROPERTY

PROPERTY bDone : BOOL
GET
bDone := m_CurMethodStates.bDone;
END_GET
END_PROPERTY

PROPERTY bError : BOOL
GET
bError := m_CurMethodStates.bError;
END_GET
SET
m_CurMethodStates.bError := bError;
END_SET
END_PROPERTY

PROPERTY bTimeout : bool
GET
bTimeout := m_tTimeoutTimer.Q;
END_GET
END_PROPERTY

PROPERTY ErrorId : WORD
GET
ErrorId := m_CurMethodStates.ErrorMsg.wErrorNo;
END_GET
SET
m_CurMethodStates.ErrorMsg.wErrorNo := ErrorId;
END_SET
END_PROPERTY

PROPERTY ErrorMsg : sErrorMsg
GET
ErrorMsg := m_CurMethodStates.ErrorMsg;
END_GET
SET
m_CurMethodStates.ErrorMsg := ErrorMsg;
END_SET
END_PROPERTY

{attribute 'object_name' := 'GoDoneState'}
METHOD GoDoneState
 m_CurMethodStates.iStateVar 	:= DONE_STATE;
 m_CurMethodStates.bDone		:= TRUE;
 m_CurMethodStates.bBusy		:= FALSE;
 
 IF NOT m_tTimeoutTimer.Q THEN
	 m_tTimeoutTimer.IN := FALSE;
	 
 END_IF
END_METHOD

{attribute 'object_name' := 'GoNextState'}
METHOD GoNextState
Inc(m_CurMethodStates.iStateVar);
END_METHOD

{attribute 'object_name' := 'GoSpecificState'}
METHOD GoSpecificState
VAR_INPUT
	iStateToJumpTo	: UINT;
END_VAR
CASE iStateToJumpTo OF
	RESET_STATE:			Reset();		
	START_STATE:			GoStartState();
	DONE_STATE:				GoDoneState();
	ELSE					m_CurMethodStates.iStateVar := iStateToJumpTo;
END_CASE
END_METHOD

METHOD PUBLIC GoStartState
VAR_INPUT
END_VAR
m_CurMethodStates.iStateVar := START_STATE;
m_CurMethodStates.bBusy		:= TRUE;
m_tTimeoutTimer.In 			:= TRUE;
END_METHOD

PROPERTY iStateVar : UINT
GET
iStateVar := m_CurMethodStates.iStateVar;
END_GET
END_PROPERTY

{attribute 'object_name' := 'Reset'}
METHOD Reset
m_CurMethodStates.bBusy 				:= FALSE;
m_CurMethodStates.bDone 				:= FALSE;
m_CurMethodStates.bError 				:= FALSE;
m_CurMethodStates.ErrorMsg.wErrorNo 	:= GVL.ERR_NO_ERROR;
m_CurMethodStates.iStateVar 			:= RESET_STATE;
m_tTimeoutTimer.In 					:= FALSE;
END_METHOD

END_FUNCTION_BLOCK

// Standard/ITF_MethodState
INTERFACE ITF_MethodState

PROPERTY bBusy : bool
GET
END_GET
END_PROPERTY

PROPERTY bDone : bool
GET
END_GET
END_PROPERTY

PROPERTY bError : bool
GET
END_GET
END_PROPERTY

PROPERTY ErrorMsg : sErrorMsg
GET
END_GET
END_PROPERTY

METHOD FINAL GoDoneState
VAR_INPUT
END_VAR
END_METHOD

METHOD FINAL GoNextState
VAR_INPUT
END_VAR
END_METHOD

METHOD FINAL GoSpecificState
VAR_INPUT
	iStateToJumpTo : UINT;
END_VAR
END_METHOD

METHOD GoStartState
VAR_INPUT
END_VAR
END_METHOD

PROPERTY iStateVar : uint
GET
END_GET
END_PROPERTY

METHOD FINAL Reset
VAR_INPUT
END_VAR
END_METHOD

END_INTERFACE

// Standard/FB_MethodState_Ext
//Author: 				Walther Ronny
//Version:				1.0
//Last change:			24.07.17
//See Release notes at the bottom
FUNCTION_BLOCK PUBLIC FB_MethodState_Ext IMPLEMENTS ITF_MethodState_Ext //Fb to help realizing a state machine inside a method
VAR_INPUT
	tTimeout : TIME;
END_VAR
VAR
	m_CurMethodStates : ST_MethodState;
	m_tTimeoutTimer : TON;
END_VAR
{library PUBLIC}
VAR CONSTANT
	RESET_STATE : UINT := 0;
	START_STATE : UINT := 1;
	DONE_STATE : UINT := 99;
END_VAR
(*
V1.0 Walther Ronny
	- initial version extended with ST_ErrorMsg
*)

m_tTimeoutTimer(PT:=tTimeout);

 IF 		m_tTimeoutTimer.Q 				//Timer eleapsed
	AND 	tTimeout <> T#0S 				//Ignore, if Timeout deactivated
	AND NOT m_CurMethodStates.bDone THEN	//Ignore, if Done set already
	
	 m_CurMethodStates.bError := TRUE;
	 GoDoneState();
	 
 END_IF

PROPERTY bBusy : BOOL
GET
bBusy := m_CurMethodStates.bBusy;
END_GET
END_PROPERTY

PROPERTY bDone : BOOL
GET
bDone := m_CurMethodStates.bDone;
END_GET
END_PROPERTY

PROPERTY bError : BOOL
GET
bError := m_CurMethodStates.bError;
END_GET
SET
m_CurMethodStates.bError := bError;
END_SET
END_PROPERTY

PROPERTY bTimeout : bool
GET
bTimeout := m_tTimeoutTimer.Q;
END_GET
END_PROPERTY

PROPERTY ErrorId : WORD
GET
ErrorId := m_CurMethodStates.ErrorMsg.wErrorNo;
END_GET
SET
m_CurMethodStates.ErrorMsg.wErrorNo := ErrorId;
END_SET
END_PROPERTY

PROPERTY ErrorMsg : ST_ErrorMsg
GET
ErrorMsg := m_CurMethodStates.ErrorMsg;
END_GET
SET
m_CurMethodStates.ErrorMsg := ErrorMsg;
END_SET
END_PROPERTY

PROPERTY ErrorType : E_ErrorTypes
GET
ErrorType := m_CurMethodStates.ErrorMsg.eErrorType;
END_GET
SET
m_CurMethodStates.ErrorMsg.eErrorType := ErrorType;
END_SET
END_PROPERTY

{attribute 'object_name' := 'GoDoneState'}
METHOD GoDoneState
 m_CurMethodStates.iStateVar 	:= DONE_STATE;
 m_CurMethodStates.bDone		:= TRUE;
 m_CurMethodStates.bBusy		:= FALSE;
 
 IF NOT m_tTimeoutTimer.Q THEN
	 m_tTimeoutTimer.IN := FALSE;
	 
 END_IF
END_METHOD

{attribute 'object_name' := 'GoNextState'}
METHOD GoNextState
Inc(m_CurMethodStates.iStateVar);
END_METHOD

{attribute 'object_name' := 'GoSpecificState'}
METHOD GoSpecificState
VAR_INPUT
	iStateToJumpTo	: UINT;
END_VAR
CASE iStateToJumpTo OF
	RESET_STATE:			Reset();		
	START_STATE:			GoStartState();
	DONE_STATE:				GoDoneState();
	ELSE					m_CurMethodStates.iStateVar := iStateToJumpTo;
END_CASE
END_METHOD

METHOD PUBLIC GoStartState
VAR_INPUT
END_VAR
m_CurMethodStates.iStateVar := START_STATE;
m_CurMethodStates.bBusy		:= TRUE;
m_tTimeoutTimer.In 			:= TRUE;
END_METHOD

PROPERTY iStateVar : UINT
GET
iStateVar := m_CurMethodStates.iStateVar;
END_GET
END_PROPERTY

{attribute 'object_name' := 'Reset'}
METHOD Reset
m_CurMethodStates.bBusy 				:= FALSE;
m_CurMethodStates.bDone 				:= FALSE;
m_CurMethodStates.bError 				:= FALSE;
m_CurMethodStates.ErrorMsg.wErrorNo 	:= GVL.ERR_NO_ERROR;
m_CurMethodStates.iStateVar 			:= RESET_STATE;
m_tTimeoutTimer.In 					:= FALSE;
END_METHOD

PROPERTY PUBLIC T_RetVal : T_RETVALUE
GET
IF m_CurMethodStates.bError THEN
	T_RetVal := eNOK;
	
ELSIF m_CurMethodStates.bDone THEN
	T_RetVal := eOK;
	
ELSE
	T_RetVal := eBUSY;
END_IF
END_GET
END_PROPERTY

END_FUNCTION_BLOCK

// Standard/ITF_MethodState_Ext
INTERFACE ITF_MethodState_Ext

PROPERTY bBusy : bool
GET
END_GET
END_PROPERTY

PROPERTY bDone : bool
GET
END_GET
END_PROPERTY

PROPERTY bError : bool
GET
END_GET
END_PROPERTY

PROPERTY ErrorMsg : ST_ErrorMsg
GET
END_GET
END_PROPERTY

METHOD FINAL GoDoneState
VAR_INPUT
END_VAR
END_METHOD

METHOD FINAL GoNextState
VAR_INPUT
END_VAR
END_METHOD

METHOD FINAL GoSpecificState
VAR_INPUT
	iStateToJumpTo : UINT;
END_VAR
END_METHOD

METHOD GoStartState
VAR_INPUT
END_VAR
END_METHOD

PROPERTY iStateVar : uint
GET
END_GET
END_PROPERTY

METHOD FINAL Reset
VAR_INPUT
END_VAR
END_METHOD

END_INTERFACE

// Standard/FB_MethodState_Ext_Data
//Author: 				Walther Ronny
//Version:				1.0
//Last change:			24.07.17
//See Release notes at the bottom
FUNCTION_BLOCK PUBLIC FB_MethodState_Ext_Data EXTENDS FB_MethodState_Ext //Fb to help realizing a state machine inside a method
VAR_INPUT
	stAdditionalData : ST_MethodState_AdditionalData;
END_VAR

(*
V1.0 Walther Ronny
	- initial version extended with ST_ErrorMsg
*)

END_FUNCTION_BLOCK

// Standard/Scale
//{attribute 'hide_all_locals'}
FUNCTION Scale : REAL //Func to scale values. Returns the scaled value
VAR_INPUT
	iX,
	iXmin,
	iXmax : INT;
	rScaleMin,
	rScaleMax : REAL;
END_VAR
VAR
	rGain,
	rOffset : REAL;
END_VAR

IF (iXmax-iXmin) <> 0 THEN
	rGain := (rScaleMax-rScaleMin)/(iXmax-iXmin);
	rOffset := (rScaleMax - rGain * iXmax);
	
	Scale := rGain * iX + rOffset;
END_IF

END_FUNCTION

// WorkstationFsm/FB_WsFsm_Base
FUNCTION_BLOCK FB_WsFsm_Base IMPLEMENTS ITF_WsFsm
VAR_INPUT
	In_bPause : BOOL;
	In_iRelDocNum :				UINT;	//Distance between previous and this WS in mm - 0 is OFF - Set just in case it is changing...!!!
END_VAR
VAR_OUTPUT
	bError_InternalStatemachine : BOOL; //Indicates an internal statemachine error, caused by an invalid transition
	
	CurrentState 	: eWsStates := eWsStates.INIT_WS;
	WsCfg 			: sWsConfiguration;
END_VAR
VAR			
	
	bProcessDocInWs 	: BOOL :=FALSE; //Flag to skip cycle if there is no document in WS at machine startup. In that case the doc pointer can be invalid!
	tTimerWsProcessing	: TON;
	pCurrentDoc			: POINTER TO sDocument;
	
	
	CurSubState 			: eSubState := eSubState.STATE_ENTRY;
	
	NextState				: eWsStates := eWsStates.UNDEFINED;
	LastStateBeforeError	: eWsStates := eWsStates.UNDEFINED;
	
	//bIsError,
	//bIsReset				: BOOL;
	bDone_tmp, bError_tmp 	: BOOL;
	DummyDocEvent : sDocEvent;
END_VAR

WsCfg.iRelDocNum := In_iRelDocNum;

CASE CurrentState OF
//======================================================================================================================================	
	eWsStates.INIT_WS : //So far, all methods here are without function. Just kept for  later use.....
				//ENTRY...................................................................
						IF CurSubState = eSubState.STATE_ENTRY THEN
							M_INIT_WS_ENTRY();
							CurSubState := eSubState.STATE_DO;													
						END_IF
				//DO......................................................................		
						IF CurSubState = eSubState.STATE_DO THEN
							M_INIT_WS_DO();
						
							IF NextState = eWsStates.IDLE OR NextState = eWsStates.ERROR THEN
								CurSubState := eSubState.STATE_EXIT;
								
							ELSIF NextState = eWsStates.UNDEFINED THEN
								//Waiting
								
							ELSE
								bError_InternalStatemachine := TRUE;	
								
							END_IF
						END_IF					
				//EXIT....................................................................	
						IF CurSubState = eSubState.STATE_EXIT THEN
							M_INIT_WS_EXIT();								
							A_DoTransition();
						END_IF	
//======================================================================================================================================	
	eWsStates.IDLE :
	
				//ENTRY...................................................................
						IF CurSubState = eSubState.STATE_ENTRY THEN
							M_IDLE_ENTRY();
							CurSubState := eSubState.STATE_DO;													
						END_IF
				//DO......................................................................		
						IF CurSubState = eSubState.STATE_DO THEN
							M_IDLE_DO();
						
							IF NextState = eWsStates.PRE_HANDLING OR NextState = eWsStates.ERROR OR NextState = eWsStates.CYCLE_FINISHED THEN
								CurSubState := eSubState.STATE_EXIT;
								
							ELSIF NextState = eWsStates.UNDEFINED THEN
								//Waiting
								
							ELSE
								bError_InternalStatemachine := TRUE;	
								
							END_IF
						END_IF					
				//EXIT....................................................................	
						IF CurSubState = eSubState.STATE_EXIT THEN
							M_IDLE_EXIT();								
							A_DoTransition();
						END_IF
//======================================================================================================================================						
	eWsStates.PRE_HANDLING :
				//ENTRY...................................................................
						IF CurSubState = eSubState.STATE_ENTRY THEN
							M_PRE_HANDLING_ENTRY();
							CurSubState := eSubState.STATE_DO;
						END_IF
				//DO......................................................................			
						IF CurSubState = eSubState.STATE_DO THEN
							M_PRE_HANDLING_DO(bDone => bDone_tmp , bError => bError_tmp);
							
							IF bDone_tmp THEN
								IF bError_tmp THEN
									NextState := eWsStates.ERROR;
								ELSE
									IF WsCfg.bVirtualWs THEN
										NextState := eWsStates.PAST_HANDLING;
									ELSE																												
										NextState := eWsStates.MASTER_SYSTEM_PROCESSING;
									END_IF	
								END_IF
								
								CurSubState := eSubState.STATE_EXIT;
								
							END_IF							
						END_IF
				//EXIT....................................................................		
						IF CurSubState = eSubState.STATE_EXIT THEN
							M_PRE_HANDLING_EXIT();
							A_DoTransition();
						END_IF
//======================================================================================================================================	
	eWsStates.MASTER_SYSTEM_PROCESSING :
				//ENTRY...................................................................
						IF CurSubState = eSubState.STATE_ENTRY THEN
							M_MASTER_SYSTEM_PROCESSING_ENTRY();
							CurSubState := eSubState.STATE_DO;													
						END_IF
				//DO......................................................................		
						IF CurSubState = eSubState.STATE_DO THEN
							M_MASTER_SYSTEM_PROCESSING_DO();
						
							IF NextState = eWsStates.PAST_HANDLING OR NextState = eWsStates.ERROR THEN
								CurSubState := eSubState.STATE_EXIT;
								
							ELSIF NextState = eWsStates.UNDEFINED THEN
								//Waiting
								
							ELSE
								bError_InternalStatemachine := TRUE;	
								
							END_IF
						END_IF
					
				//EXIT....................................................................	
						IF CurSubState = eSubState.STATE_EXIT THEN
							M_MASTER_SYSTEM_PROCESSING_EXIT();								
							A_DoTransition();
						END_IF
//======================================================================================================================================						
	eWsStates.PAST_HANDLING :
	
				//ENTRY...................................................................
						IF CurSubState = eSubState.STATE_ENTRY THEN
							M_PAST_HANDLING_ENTRY();
							CurSubState := eSubState.STATE_DO;
						END_IF
				//DO......................................................................		
						IF CurSubState = eSubState.STATE_DO THEN
							M_PAST_HANDLING_DO(bDone => bDone_tmp , bError => bError_tmp);
							
							IF bDone_tmp THEN
								IF bError_tmp THEN
									NextState := eWsStates.ERROR;
								ELSE
									NextState := eWsStates.CYCLE_FINISHED;	
								END_IF
								
								CurSubState := eSubState.STATE_EXIT;
								
							END_IF								
						END_IF
				//EXIT....................................................................		
						IF CurSubState = eSubState.STATE_EXIT THEN
							M_PAST_HANDLING_EXIT();
							A_DoTransition();
						END_IF
//======================================================================================================================================						
	eWsStates.CYCLE_FINISHED :
				//ENTRY...................................................................
						IF CurSubState = eSubState.STATE_ENTRY THEN
							M_CYCLE_FINISHED_ENTRY();
							CurSubState := eSubState.STATE_DO;
						END_IF
				//DO......................................................................			
						IF CurSubState = eSubState.STATE_DO THEN
							M_CYCLE_FINISHED_DO();
							
							IF NextState = eWsStates.IDLE OR NextState = eWsStates.ERROR THEN
								CurSubState := eSubState.STATE_EXIT;
								
							END_IF							
						END_IF
				//EXIT....................................................................			
						IF CurSubState = eSubState.STATE_EXIT THEN
							M_CYCLE_FINISHED_EXIT();
							A_DoTransition();
						END_IF
//======================================================================================================================================						
	eWsStates.ERROR :
				//ENTRY...................................................................
						IF CurSubState = eSubState.STATE_ENTRY THEN
							M_CYCLE_FINISHED_ENTRY();
							CurSubState := eSubState.STATE_DO;
						END_IF
				//DO......................................................................			
						IF CurSubState = eSubState.STATE_DO THEN
							M_ERROR_DO();
							
							IF NextState = eWsStates.IDLE OR NextState = eWsStates.ERROR OR CurrentState = eWsStates.WS_PROCESSING THEN
								CurSubState := eSubState.STATE_EXIT;
								
							END_IF							
						END_IF
				//EXIT....................................................................			
						IF CurSubState = eSubState.STATE_EXIT THEN
							M_ERROR_EXIT();
							CurSubState := eSubState.STATE_ENTRY;
						END_IF
//======================================================================================================================================	
END_CASE

ACTION A_DoTransition:
LastStateBeforeError := eWsStates.UNDEFINED;

IF NextState = eWsStates.ERROR THEN
	LastStateBeforeError := CurrentState;
	
	M_WS_PROCESSING_INTO_ERROR();
	
END_IF

CurrentState 	:= NextState;
NextState 		:= eWsStates.UNDEFINED;
CurSubState 	:= eSubState.STATE_ENTRY;
END_ACTION

METHOD FB_init : bool
VAR_INPUT
	bInitRetains 			: BOOL; 															// if TRUE, the retain variables are initialized (warm start / cold start)
	bInCopyCode 			: BOOL;  															// if TRUE, the instance afterwards gets moved into the copy code (online change)
	
	iWsNum : 				UINT;
	iRelDocNum :				UINT;	//Distance between previous and this WS in mm - 0 is OFF
	iLocation :					UINT;		
	bVirtualWs : 				BOOL;
	tWsProcessingTimeout :		TIME;	//Timeout for composite state WsProcessing
	OperationType: 				eWsOperationType;
	
	pEvt_DocIn, 
	pEvt_DocProcessStart,
	pEvt_DocOut : 				POINTER TO sDocEvent;
	
	wCompId : 					WORD;
	
	//Document will be unlocked when method M_FinishCycle is called. 
	//Flag shall be set to TRUE, if Ws is the last WS to enable the host to remove the doc from the buffer
	bUnlockDocAtFinishing : BOOL; 
END_VAR
WsCfg.iWsNum 				:= iWsNum;
WsCfg.iRelDocNum 			:= iRelDocNum;
WsCfg.iLocation 			:= iLocation;		
WsCfg.bVirtualWs 			:= bVirtualWs;
WsCfg.tWsProcessingTimeout 	:= tWsProcessingTimeout;
WsCfg.OperationType 		:= OperationType;
WsCfg.bUnlockDocAtFinishing := bUnlockDocAtFinishing;

In_iRelDocNum := iRelDocNum;

IF IsValidPtr(pEvt_DocIn) THEN	
	WsCfg.pEvt_DocIn 			:= pEvt_DocIn;
	WsCfg.bEvt_DocIn_WasSet		:= TRUE;
ELSE
	WsCfg.pEvt_DocIn 			:= ADR(DummyDocEvent);;
	WsCfg.bEvt_DocIn_WasSet		:= FALSE;	
END_IF

IF IsValidPtr(pEvt_DocProcessStart) THEN	
	WsCfg.pEvt_DocProcessStart 			:= pEvt_DocProcessStart;
	WsCfg.pEvt_DocProcessStart_WasSet	:= TRUE;
ELSE
	WsCfg.pEvt_DocProcessStart 			:= ADR(DummyDocEvent);;
	WsCfg.pEvt_DocProcessStart_WasSet	:= FALSE;	
END_IF

IF IsValidPtr(pEvt_DocOut) THEN	
	WsCfg.pEvt_DocOut 			:= pEvt_DocOut;
	WsCfg.pEvt_DocOut_wasSet	:= TRUE;
ELSE
	WsCfg.pEvt_DocOut 			:= ADR(DummyDocEvent);;
	WsCfg.pEvt_DocOut_wasSet	:= FALSE;	
END_IF

WsCfg.wCompId 				:= wCompId;
END_METHOD

METHOD PRIVATE M_ThrowError
VAR_INPUT
	SrcState : eWsStates;
	ErrorMsg : sErrorMsg;
END_VAR
ErrorMsg.sFunctionName := CONCAT('FB_WsFsm.', ErrorMsg.sFunctionName);
ErrorManagement.M_InsertNewError(ErrorMsg := ErrorMsg);
END_METHOD

METHOD M_ERROR_DO //can be derived in order to add own code
END_METHOD

METHOD M_PAST_HANDLING_DO //can be derived in order to add own code
VAR_OUTPUT
	bDone,
	bError : BOOL;
END_VAR
bDone := TRUE;
END_METHOD

METHOD M_PAST_HANDLING_ENTRY //can be derived in order to add own code
END_METHOD

METHOD M_PAST_HANDLING_EXIT //can be derived in order to add own code
END_METHOD

METHOD M_PRE_HANDLING_DO //can be derived in order to add own code
VAR_OUTPUT
	bDone,
	bError : BOOL;
END_VAR
bDone := TRUE;
END_METHOD

METHOD M_PRE_HANDLING_ENTRY //can be derived in order to add own code
END_METHOD

METHOD M_PRE_HANDLING_EXIT //can be derived in order to add own code
END_METHOD

METHOD PUBLIC M_FinishCycle : bool
VAR
	LogMsg : STRING ;
	Evt_DocOut : sDocEvent;
	bMethodError: BOOL := FALSE;
	MethodErrorMsg: sErrorMsg;
END_VAR
MethodErrorMsg.sFunctionName 	:= 'M_FinishCycle';
MethodErrorMsg.wComponent 		:= WsCfg.wCompId;

IF CurrentState = eWsStates.CYCLE_FINISHED THEN
		
	IF IsValidPtr(pCurrentDoc) AND bProcessDocInWs THEN		//Document was processed before, so set doc array parameter and send doc_out event
		//Set doc to  moving thus leaving WS
			pCurrentDoc^.Moving := TRUE;
			
		//Set following location
			pCurrentDoc^.Location := WsCfg.iLocation+1;
			
		//UnLock document if configured
		IF WsCfg.bUnlockDocAtFinishing THEN
			pCurrentDoc^.bLockedBySps := FALSE;
		END_IF
		
		//Generate OK Event
			Evt_DocOut.DocID := pCurrentDoc^.ID;
			Evt_DocOut.EventChangeFlag := switch(WsCfg.pEvt_DocOut^.EventChangeFlag);
				
			WsCfg.pEvt_DocOut^ := Evt_DocOut;
			
		//switch to next state
			NextState := eWsStates.IDLE;
			
		IF GVL_Statemachine_ERROR_IDS.bLoggingOnOff THEN	
			//Logging Doc Event	
			LogMsg := CONCAT('|CompId: ', WORD_TO_STRING(WsCfg.wCompId));
			LogMsg := CONCAT(LogMsg, '|WsNum: ');
			LogMsg := CONCAT(LogMsg, UINT_TO_STRING(WsCfg.iWsNum));
			LogMsg := CONCAT(LogMsg,'|DocOut Event written with DocId ');
			LogMsg := CONCAT(LogMsg, UDINT_TO_STRING(WsCfg.pEvt_DocOut^.DocID));
			Logging.Debug('FB_WsFsm.M_FinishCycle', LogMsg);					

